LIN {X 0,Y 573.251,Z 441.775,A -85,B 0,C 180,E1 -2241.895,E2 -2241.895} C_VEL
LIN {X 0,Y 573.192,Z 450.436,A -85,B 0,C 180,E1 -2242.603,E2 -2242.603} C_VEL
LIN {X 0,Y 573.159,Z 458.426,A -85,B 0,C 180,E1 -2243.424,E2 -2243.424} C_VEL
LIN {X 0,Y 573.113,Z 464.437,A -85,B 0,C 180,E1 -2244.194,E2 -2244.194} C_VEL
LIN {X 0,Y 572.995,Z 469.99,A -85,B 0,C 180,E1 -2245.075,E2 -2245.075} C_VEL
LIN {X 0,Y 573.036,Z 475.15,A -85,B 0,C 180,E1 -2246.133,E2 -2246.133} C_VEL
LIN {X 0,Y 572.99,Z 477.789,A -85,B 0,C 180,E1 -2246.836,E2 -2246.836} C_VEL
LIN {X 0,Y 572.94,Z 480.683,A -85,B 0,C 180,E1 -2247.891,E2 -2247.891} C_VEL
LIN {X 0,Y 572.944,Z 481.935,A -85,B 0,C 180,E1 -2248.595,E2 -2248.595} C_VEL
LIN {X 0,Y 572.937,Z 482.71,A -85,B 0,C 180,E1 -2249.298,E2 -2249.298} C_VEL
LIN {X 0,Y 572.935,Z 483,A -85,B 0,C 180,E1 -2250,E2 -2250} C_VEL
LIN {X 0,Y 572.937,Z 482.709,A -85,B 0,C 180,E1 -2250.703,E2 -2250.703} C_VEL
LIN {X 0,Y 572.944,Z 481.934,A -85,B 0,C 180,E1 -2251.406,E2 -2251.406} C_VEL
LIN {X 0,Y 572.94,Z 480.68,A -85,B 0,C 180,E1 -2252.109,E2 -2252.109} C_VEL
LIN {X 0,Y 572.99,Z 477.786,A -85,B 0,C 180,E1 -2253.164,E2 -2253.164} C_VEL
LIN {X 0,Y 573.036,Z 475.147,A -85,B 0,C 180,E1 -2253.868,E2 -2253.868} C_VEL
LIN {X 0,Y 572.995,Z 469.984,A -85,B 0,C 180,E1 -2254.926,E2 -2254.926} C_VEL
LIN {X 0,Y 573.138,Z 463.183,A -85,B 0,C 180,E1 -2255.983,E2 -2255.983} C_VEL
LIN {X 0,Y 573.164,Z 455.8,A -85,B 0,C 180,E1 -2256.86,E2 -2256.86} C_VEL
LIN {X 0,Y 573.215,Z 448.402,A -85,B 0,C 180,E1 -2257.574,E2 -2257.574} C_VEL
LIN {X 0,Y 573.278,Z 440.539,A -85,B 0,C 180,E1 -2258.194,E2 -2258.194} C_VEL
LIN {X 0,Y 573.323,Z 430.724,A -85,B 0,C 180,E1 -2258.814,E2 -2258.814} C_VEL
LIN {X 0,Y 573.387,Z 419.295,A -85,B 0,C 180,E1 -2259.347,E2 -2259.347} C_VEL
LIN {X 0,Y 573.48,Z 409.234,A -85,B 0,C 180,E1 -2259.679,E2 -2259.679} C_VEL
LIN {X 0,Y 573.512,Z 400.423,A -85,B 0,C 180,E1 -2259.879,E2 -2259.879} C_VEL
LIN {X 0,Y 573.604,Z 327.515,A -85,B 0,C 180,E1 -2260.808,E2 -2260.808} C_VEL
LIN {X 0,Y 573.152,Z 322.288,A -85,B 0,C 180,E1 -2260.89,E2 -2260.89} C_VEL
LIN {X 0,Y 573.327,Z 305.23,A -85,B 0,C 180,E1 -2263.469,E2 -2263.469} C_VEL
LIN {X 0,Y 573.462,Z 287.427,A -85,B 0,C 180,E1 -2266.189,E2 -2266.189} C_VEL
LIN {X 0,Y 573.63,Z 269.625,A -85,B 0,C 180,E1 -2268.946,E2 -2268.946} C_VEL
LIN {X 0,Y 573.779,Z 252.639,A -85,B 0,C 180,E1 -2271.559,E2 -2271.559} C_VEL
LIN {X 0,Y 573.655,Z 246.517,A -85,B 0,C 180,E1 -2272.511,E2 -2272.511} C_VEL
LIN {X 0,Y 573.209,Z 243.899,A -85,B 0,C 180,E1 -2272.946,E2 -2272.946} C_VEL
LIN {X 0,Y 573.2,Z 243.901,A -85,B 0,C 180,E1 -2275.413,E2 -2275.413} C_VEL
LIN {X 0,Y 573.191,Z 243.894,A -85,B 0,C 180,E1 -2278.018,E2 -2278.018} C_VEL
LIN {X 0,Y 573.2,Z 243.895,A -85,B 0,C 180,E1 -2280.877,E2 -2280.877} C_VEL
LIN {X 0,Y 573.215,Z 243.896,A -85,B 0,C 180,E1 -2283.517,E2 -2283.517} C_VEL
LIN {X 0,Y 573.176,Z 243.895,A -85,B 0,C 180,E1 -2286.055,E2 -2286.055} C_VEL
LIN {X 0,Y 573.175,Z 243.898,A -85,B 0,C 180,E1 -2288.707,E2 -2288.707} C_VEL
LIN {X 0,Y 573.19,Z 243.896,A -85,B 0,C 180,E1 -2291.588,E2 -2291.588} C_VEL
LIN {X 0,Y 573.204,Z 243.896,A -85,B 0,C 180,E1 -2294.673,E2 -2294.673} C_VEL
LIN {X 0,Y 573.2,Z 243.893,A -85,B 0,C 180,E1 -2297.596,E2 -2297.596} C_VEL
LIN {X 0,Y 573.229,Z 243.893,A -85,B 0,C 180,E1 -2300.57,E2 -2300.57} C_VEL
LIN {X 0,Y 573.219,Z 243.896,A -85,B 0,C 180,E1 -2303.075,E2 -2303.075} C_VEL
LIN {X 0,Y 573.232,Z 243.888,A -85,B 0,C 180,E1 -2305.669,E2 -2305.669} C_VEL
LIN {X 0,Y 573.205,Z 243.893,A -85,B 0,C 180,E1 -2308.182,E2 -2308.182} C_VEL
LIN {X 0,Y 573.212,Z 243.899,A -85,B 0,C 180,E1 -2310.631,E2 -2310.631} C_VEL
LIN {X 0,Y 573.194,Z 243.893,A -85,B 0,C 180,E1 -2313.517,E2 -2313.517} C_VEL
LIN {X 0,Y 573.188,Z 243.897,A -85,B 0,C 180,E1 -2316.133,E2 -2316.133} C_VEL
LIN {X 0,Y 573.216,Z 243.892,A -85,B 0,C 180,E1 -2319.172,E2 -2319.172} C_VEL
LIN {X 0,Y 573.195,Z 243.898,A -85,B 0,C 180,E1 -2322.15,E2 -2322.15} C_VEL
LIN {X 0,Y 573.209,Z 243.892,A -85,B 0,C 180,E1 -2325.08,E2 -2325.08} C_VEL
LIN {X 0,Y 573.223,Z 243.893,A -85,B 0,C 180,E1 -2327.97,E2 -2327.97} C_VEL
LIN {X 0,Y 573.2,Z 243.899,A -85,B 0,C 180,E1 -2330.116,E2 -2330.116} C_VEL
LIN {X 0,Y 573.221,Z 243.891,A -85,B 0,C 180,E1 -2332.958,E2 -2332.958} C_VEL
LIN {X 0,Y 573.271,Z 243.884,A -85,B 0,C 180,E1 -2335.077,E2 -2335.077} C_VEL
LIN {X 0,Y 573.307,Z 243.885,A -85,B 0,C 180,E1 -2337.892,E2 -2337.892} C_VEL
LIN {X 0,Y 573.316,Z 243.886,A -85,B 0,C 180,E1 -2340,E2 -2340} C_VEL
LIN {X 0,Y 573.27,Z 243.884,A -85,B 0,C 180,E1 -2342.811,E2 -2342.811} C_VEL
LIN {X 0,Y 573.265,Z 243.888,A -85,B 0,C 180,E1 -2345.629,E2 -2345.629} C_VEL
LIN {X 0,Y 573.234,Z 243.891,A -85,B 0,C 180,E1 -2348.46,E2 -2348.46} C_VEL
LIN {X 0,Y 573.236,Z 243.89,A -85,B 0,C 180,E1 -2351.313,E2 -2351.313} C_VEL
LIN {X 0,Y 573.238,Z 243.89,A -85,B 0,C 180,E1 -2354.406,E2 -2354.406} C_VEL
LIN {X 0,Y 573.193,Z 243.895,A -85,B 0,C 180,E1 -2357.114,E2 -2357.114} C_VEL
LIN {X 0,Y 573.204,Z 243.896,A -85,B 0,C 180,E1 -2360.078,E2 -2360.078} C_VEL
LIN {X 0,Y 573.195,Z 243.894,A -85,B 0,C 180,E1 -2362.34,E2 -2362.34} C_VEL
LIN {X 0,Y 573.194,Z 243.894,A -85,B 0,C 180,E1 -2364.344,E2 -2364.344} C_VEL
LIN {X 0,Y 572.557,Z 243.974,A -85,B 0,C 180,E1 -2364.93,E2 -2364.93} C_VEL
LIN {X 0,Y 569.725,Z 244.332,A -85,B 0,C 180,E1 -2365.882,E2 -2365.882} C_VEL
LIN {X 0,Y 567.305,Z 244.636,A -85,B 0,C 180,E1 -2366.647,E2 -2366.647} C_VEL
LIN {X 0,Y 566.246,Z 244.766,A -85,B 0,C 180,E1 -2367.238,E2 -2367.238} C_VEL
LIN {X 0,Y 566.151,Z 244.776,A -85,B 0,C 180,E1 -2367.439,E2 -2367.439} C_VEL
LIN {X 0,Y 566.149,Z 244.777,A -85,B 0,C 180,E1 -2369.772,E2 -2369.772} C_VEL
LIN {X 0,Y 566.192,Z 244.766,A -85,B 0,C 180,E1 -2372.428,E2 -2372.428} C_VEL
LIN {X 0,Y 566.164,Z 244.773,A -85,B 0,C 180,E1 -2374.987,E2 -2374.987} C_VEL
LIN {X 0,Y 566.189,Z 244.774,A -85,B 0,C 180,E1 -2377.462,E2 -2377.462} C_VEL
LIN {X 0,Y 566.195,Z 244.765,A -85,B 0,C 180,E1 -2380.2,E2 -2380.2} C_VEL
LIN {X 0,Y 566.179,Z 244.774,A -85,B 0,C 180,E1 -2383.056,E2 -2383.056} C_VEL
LIN {X 0,Y 566.156,Z 244.77,A -85,B 0,C 180,E1 -2386.053,E2 -2386.053} C_VEL
LIN {X 0,Y 566.155,Z 244.776,A -85,B 0,C 180,E1 -2388.858,E2 -2388.858} C_VEL
LIN {X 0,Y 566.203,Z 244.768,A -85,B 0,C 180,E1 -2391.443,E2 -2391.443} C_VEL
LIN {X 0,Y 566.141,Z 244.773,A -85,B 0,C 180,E1 -2394.306,E2 -2394.306} C_VEL
LIN {X 0,Y 566.194,Z 244.773,A -85,B 0,C 180,E1 -2396.896,E2 -2396.896} C_VEL
LIN {X 0,Y 566.16,Z 244.772,A -85,B 0,C 180,E1 -2399.406,E2 -2399.406} C_VEL
LIN {X 0,Y 566.149,Z 244.771,A -85,B 0,C 180,E1 -2401.854,E2 -2401.854} C_VEL
LIN {X 0,Y 566.187,Z 244.768,A -85,B 0,C 180,E1 -2404.249,E2 -2404.249} C_VEL
LIN {X 0,Y 566.147,Z 244.773,A -85,B 0,C 180,E1 -2407.367,E2 -2407.367} C_VEL
LIN {X 0,Y 566.171,Z 244.768,A -85,B 0,C 180,E1 -2409.661,E2 -2409.661} C_VEL
LIN {X 0,Y 566.166,Z 244.769,A -85,B 0,C 180,E1 -2411.92,E2 -2411.92} C_VEL
LIN {X 0,Y 566.172,Z 244.839,A -85,B 0,C 180,E1 -2414.198,E2 -2414.198} C_VEL
LIN {X 0,Y 566.045,Z 256.904,A -85,B 0,C 180,E1 -2417.086,E2 -2417.086} C_VEL
LIN {X 0,Y 565.985,Z 265.442,A -85,B 0,C 180,E1 -2419.063,E2 -2419.063} C_VEL
LIN {X 0,Y 566.666,Z 271.419,A -85,B 0,C 180,E1 -2419.152,E2 -2419.152} C_VEL
LIN {X 0,Y 566.539,Z 340.424,A -85,B 0,C 180,E1 -2420.043,E2 -2420.043} C_VEL
LIN {X 0,Y 566.455,Z 350.067,A -85,B 0,C 180,E1 -2420.267,E2 -2420.267} C_VEL
LIN {X 0,Y 566.371,Z 361.605,A -85,B 0,C 180,E1 -2420.671,E2 -2420.671} C_VEL
LIN {X 0,Y 566.299,Z 371.47,A -85,B 0,C 180,E1 -2421.165,E2 -2421.165} C_VEL
LIN {X 0,Y 566.252,Z 379.918,A -85,B 0,C 180,E1 -2421.704,E2 -2421.704} C_VEL
LIN {X 0,Y 566.169,Z 387.886,A -85,B 0,C 180,E1 -2422.331,E2 -2422.331} C_VEL
LIN {X 0,Y 566.099,Z 394.656,A -85,B 0,C 180,E1 -2422.978,E2 -2422.978} C_VEL
LIN {X 0,Y 566.071,Z 399.998,A -85,B 0,C 180,E1 -2423.584,E2 -2423.584} C_VEL
LIN {X 0,Y 566.025,Z 405.309,A -85,B 0,C 180,E1 -2424.299,E2 -2424.299} C_VEL
LIN {X 0,Y 565.917,Z 409.743,A -85,B 0,C 180,E1 -2425.013,E2 -2425.013} C_VEL
LIN {X 0,Y 565.961,Z 413.439,A -85,B 0,C 180,E1 -2425.727,E2 -2425.727} C_VEL
LIN {X 0,Y 565.914,Z 417.641,A -85,B 0,C 180,E1 -2426.796,E2 -2426.796} C_VEL
LIN {X 0,Y 565.842,Z 420.579,A -85,B 0,C 180,E1 -2427.864,E2 -2427.864} C_VEL
LIN {X 0,Y 565.844,Z 421.871,A -85,B 0,C 180,E1 -2428.576,E2 -2428.576} C_VEL
LIN {X 0,Y 565.837,Z 422.688,A -85,B 0,C 180,E1 -2429.288,E2 -2429.288} C_VEL
LIN {X 0,Y 565.837,Z 422.996,A -85,B 0,C 180,E1 -2430,E2 -2430} C_VEL
LIN {X 0,Y 565.838,Z 422.729,A -85,B 0,C 180,E1 -2430.711,E2 -2430.711} C_VEL
LIN {X 0,Y 565.845,Z 421.994,A -85,B 0,C 180,E1 -2431.423,E2 -2431.423} C_VEL
LIN {X 0,Y 565.842,Z 420.785,A -85,B 0,C 180,E1 -2432.135,E2 -2432.135} C_VEL
LIN {X 0,Y 565.913,Z 417.934,A -85,B 0,C 180,E1 -2433.203,E2 -2433.203} C_VEL
LIN {X 0,Y 565.935,Z 415.342,A -85,B 0,C 180,E1 -2433.916,E2 -2433.916} C_VEL
LIN {X 0,Y 565.895,Z 410.232,A -85,B 0,C 180,E1 -2434.987,E2 -2434.987} C_VEL
LIN {X 0,Y 566.057,Z 404.734,A -85,B 0,C 180,E1 -2435.879,E2 -2435.879} C_VEL
LIN {X 0,Y 566.077,Z 397.824,A -85,B 0,C 180,E1 -2436.775,E2 -2436.775} C_VEL
LIN {X 0,Y 566.149,Z 388.913,A -85,B 0,C 180,E1 -2437.668,E2 -2437.668} C_VEL
LIN {X 0,Y 566.267,Z 381.158,A -85,B 0,C 180,E1 -2438.295,E2 -2438.295} C_VEL
LIN {X 0,Y 566.32,Z 372.983,A -85,B 0,C 180,E1 -2438.834,E2 -2438.834} C_VEL
LIN {X 0,Y 566.342,Z 364.464,A -85,B 0,C 180,E1 -2439.283,E2 -2439.283} C_VEL
LIN {X 0,Y 566.439,Z 353.233,A -85,B 0,C 180,E1 -2439.732,E2 -2439.732} C_VEL
LIN {X 0,Y 566.573,Z 341.753,A -85,B 0,C 180,E1 -2440.023,E2 -2440.023} C_VEL
LIN {X 0,Y 566.601,Z 322.559,A -85,B 0,C 180,E1 -2440.293,E2 -2440.293} C_VEL
LIN {X 0,Y 566.545,Z 269.375,A -85,B 0,C 180,E1 -2440.966,E2 -2440.966} C_VEL
LIN {X 0,Y 565.964,Z 265.144,A -85,B 0,C 180,E1 -2441.048,E2 -2441.048} C_VEL
LIN {X 0,Y 566.063,Z 254.223,A -85,B 0,C 180,E1 -2443.644,E2 -2443.644} C_VEL
LIN {X 0,Y 566.154,Z 244.775,A -85,B 0,C 180,E1 -2445.941,E2 -2445.941} C_VEL
LIN {X 0,Y 566.181,Z 244.768,A -85,B 0,C 180,E1 -2448.828,E2 -2448.828} C_VEL
LIN {X 0,Y 566.193,Z 244.773,A -85,B 0,C 180,E1 -2451.416,E2 -2451.416} C_VEL
LIN {X 0,Y 566.151,Z 244.771,A -85,B 0,C 180,E1 -2454.182,E2 -2454.182} C_VEL
LIN {X 0,Y 566.173,Z 244.77,A -85,B 0,C 180,E1 -2456.652,E2 -2456.652} C_VEL
LIN {X 0,Y 566.147,Z 244.773,A -85,B 0,C 180,E1 -2459.771,E2 -2459.771} C_VEL
LIN {X 0,Y 566.188,Z 244.767,A -85,B 0,C 180,E1 -2462.427,E2 -2462.427} C_VEL
LIN {X 0,Y 566.158,Z 244.778,A -85,B 0,C 180,E1 -2464.986,E2 -2464.986} C_VEL
LIN {X 0,Y 566.187,Z 244.77,A -85,B 0,C 180,E1 -2467.461,E2 -2467.461} C_VEL
LIN {X 0,Y 566.201,Z 244.765,A -85,B 0,C 180,E1 -2470.199,E2 -2470.199} C_VEL
LIN {X 0,Y 566.174,Z 244.776,A -85,B 0,C 180,E1 -2473.056,E2 -2473.056} C_VEL
LIN {X 0,Y 566.151,Z 244.771,A -85,B 0,C 180,E1 -2476.053,E2 -2476.053} C_VEL
LIN {X 0,Y 566.145,Z 244.779,A -85,B 0,C 180,E1 -2478.858,E2 -2478.858} C_VEL
LIN {X 0,Y 566.193,Z 244.766,A -85,B 0,C 180,E1 -2481.443,E2 -2481.443} C_VEL
LIN {X 0,Y 566.134,Z 244.777,A -85,B 0,C 180,E1 -2484.306,E2 -2484.306} C_VEL
LIN {X 0,Y 566.187,Z 244.772,A -85,B 0,C 180,E1 -2486.896,E2 -2486.896} C_VEL
LIN {X 0,Y 566.154,Z 244.771,A -85,B 0,C 180,E1 -2489.406,E2 -2489.406} C_VEL
LIN {X 0,Y 566.136,Z 244.774,A -85,B 0,C 180,E1 -2491.853,E2 -2491.853} C_VEL
LIN {X 0,Y 566.183,Z 244.773,A -85,B 0,C 180,E1 -2494.249,E2 -2494.249} C_VEL
LIN {X 0,Y 566.15,Z 244.776,A -85,B 0,C 180,E1 -2496.722,E2 -2496.722} C_VEL
LIN {X 0,Y 566.184,Z 244.769,A -85,B 0,C 180,E1 -2498.901,E2 -2498.901} C_VEL
LIN {X 0,Y 566.176,Z 244.768,A -85,B 0,C 180,E1 -2501.171,E2 -2501.171} C_VEL
LIN {X 0,Y 566.163,Z 244.777,A -85,B 0,C 180,E1 -2504.151,E2 -2504.151} C_VEL
LIN {X 0,Y 566.156,Z 244.778,A -85,B 0,C 180,E1 -2506.358,E2 -2506.358} C_VEL
LIN {X 0,Y 566.205,Z 244.764,A -85,B 0,C 180,E1 -2509.27,E2 -2509.27} C_VEL
LIN {X 0,Y 566.181,Z 244.775,A -85,B 0,C 180,E1 -2512.152,E2 -2512.152} C_VEL
LIN {X 0,Y 566.244,Z 244.759,A -85,B 0,C 180,E1 -2515.016,E2 -2515.016} C_VEL
LIN {X 0,Y 566.274,Z 244.763,A -85,B 0,C 180,E1 -2517.866,E2 -2517.866} C_VEL
LIN {X 0,Y 566.28,Z 244.763,A -85,B 0,C 180,E1 -2520,E2 -2520} C_VEL
LIN {X 0,Y 566.231,Z 244.761,A -85,B 0,C 180,E1 -2522.846,E2 -2522.846} C_VEL
LIN {X 0,Y 566.232,Z 244.768,A -85,B 0,C 180,E1 -2525.699,E2 -2525.699} C_VEL
LIN {X 0,Y 566.179,Z 244.767,A -85,B 0,C 180,E1 -2528.566,E2 -2528.566} C_VEL
LIN {X 0,Y 566.186,Z 244.772,A -85,B 0,C 180,E1 -2531.455,E2 -2531.455} C_VEL
LIN {X 0,Y 566.196,Z 244.765,A -85,B 0,C 180,E1 -2534.494,E2 -2534.494} C_VEL
LIN {X 0,Y 566.15,Z 244.777,A -85,B 0,C 180,E1 -2537.333,E2 -2537.333} C_VEL
LIN {X 0,Y 566.167,Z 244.777,A -85,B 0,C 180,E1 -2539.582,E2 -2539.582} C_VEL
LIN {X 0,Y 566.14,Z 244.776,A -85,B 0,C 180,E1 -2541.865,E2 -2541.865} C_VEL
LIN {X 0,Y 566.145,Z 244.772,A -85,B 0,C 180,E1 -2544.183,E2 -2544.183} C_VEL
LIN {X 0,Y 566.164,Z 244.77,A -85,B 0,C 180,E1 -2546.652,E2 -2546.652} C_VEL
LIN {X 0,Y 566.14,Z 244.775,A -85,B 0,C 180,E1 -2549.772,E2 -2549.772} C_VEL
LIN {X 0,Y 566.184,Z 244.767,A -85,B 0,C 180,E1 -2552.428,E2 -2552.428} C_VEL
LIN {X 0,Y 566.153,Z 244.777,A -85,B 0,C 180,E1 -2554.986,E2 -2554.986} C_VEL
LIN {X 0,Y 566.182,Z 244.771,A -85,B 0,C 180,E1 -2557.462,E2 -2557.462} C_VEL
LIN {X 0,Y 566.16,Z 244.769,A -85,B 0,C 180,E1 -2560.203,E2 -2560.203} C_VEL
LIN {X 0,Y 566.17,Z 244.777,A -85,B 0,C 180,E1 -2563.057,E2 -2563.057} C_VEL
LIN {X 0,Y 566.149,Z 244.77,A -85,B 0,C 180,E1 -2566.054,E2 -2566.054} C_VEL
LIN {X 0,Y 566.139,Z 244.78,A -85,B 0,C 180,E1 -2568.858,E2 -2568.858} C_VEL
LIN {X 0,Y 566.165,Z 244.769,A -85,B 0,C 180,E1 -2571.636,E2 -2571.636} C_VEL
LIN {X 0,Y 566.125,Z 244.776,A -85,B 0,C 180,E1 -2574.306,E2 -2574.306} C_VEL
LIN {X 0,Y 566.156,Z 244.776,A -85,B 0,C 180,E1 -2576.894,E2 -2576.894} C_VEL
LIN {X 0,Y 566.144,Z 244.771,A -85,B 0,C 180,E1 -2579.406,E2 -2579.406} C_VEL
LIN {X 0,Y 566.135,Z 244.773,A -85,B 0,C 180,E1 -2581.854,E2 -2581.854} C_VEL
LIN {X 0,Y 566.167,Z 244.773,A -85,B 0,C 180,E1 -2584.249,E2 -2584.249} C_VEL
LIN {X 0,Y 566.163,Z 244.885,A -85,B 0,C 180,E1 -2586.982,E2 -2586.982} C_VEL
LIN {X 0,Y 566.811,Z 249.814,A -85,B 0,C 180,E1 -2587.78,E2 -2587.78} C_VEL
LIN {X 0,Y 566.655,Z 267.933,A -85,B 0,C 180,E1 -2590.595,E2 -2590.595} C_VEL
LIN {X 0,Y 566.529,Z 284.237,A -85,B 0,C 180,E1 -2593.108,E2 -2593.108} C_VEL
LIN {X 0,Y 566.343,Z 304.048,A -85,B 0,C 180,E1 -2596.18,E2 -2596.18} C_VEL
LIN {X 0,Y 566.126,Z 322.264,A -85,B 0,C 180,E1 -2598.97,E2 -2598.97} C_VEL
LIN {X 0,Y 566.684,Z 329.654,A -85,B 0,C 180,E1 -2599.085,E2 -2599.085} C_VEL
LIN {X 0,Y 566.566,Z 399.163,A -85,B 0,C 180,E1 -2599.977,E2 -2599.977} C_VEL
LIN {X 0,Y 566.464,Z 408.427,A -85,B 0,C 180,E1 -2600.178,E2 -2600.178} C_VEL
LIN {X 0,Y 566.416,Z 416.898,A -85,B 0,C 180,E1 -2600.448,E2 -2600.448} C_VEL
LIN {X 0,Y 566.336,Z 425.403,A -85,B 0,C 180,E1 -2600.807,E2 -2600.807} C_VEL
LIN {X 0,Y 566.317,Z 433.734,A -85,B 0,C 180,E1 -2601.256,E2 -2601.256} C_VEL
LIN {X 0,Y 566.211,Z 441.772,A -85,B 0,C 180,E1 -2601.794,E2 -2601.794} C_VEL
LIN {X 0,Y 566.126,Z 450.436,A -85,B 0,C 180,E1 -2602.511,E2 -2602.511} C_VEL
LIN {X 0,Y 566.087,Z 458.905,A -85,B 0,C 180,E1 -2603.402,E2 -2603.402} C_VEL
LIN {X 0,Y 566.057,Z 464.438,A -85,B 0,C 180,E1 -2604.121,E2 -2604.121} C_VEL
LIN {X 0,Y 565.906,Z 469.991,A -85,B 0,C 180,E1 -2605.013,E2 -2605.013} C_VEL
LIN {X 0,Y 565.943,Z 475.15,A -85,B 0,C 180,E1 -2606.084,E2 -2606.084} C_VEL
LIN {X 0,Y 565.88,Z 478.937,A -85,B 0,C 180,E1 -2607.153,E2 -2607.153} C_VEL
LIN {X 0,Y 565.841,Z 480.683,A -85,B 0,C 180,E1 -2607.865,E2 -2607.865} C_VEL
LIN {X 0,Y 565.844,Z 481.934,A -85,B 0,C 180,E1 -2608.577,E2 -2608.577} C_VEL
LIN {X 0,Y 565.837,Z 482.709,A -85,B 0,C 180,E1 -2609.289,E2 -2609.289} C_VEL
LIN {X 0,Y 565.836,Z 483,A -85,B 0,C 180,E1 -2610,E2 -2610} C_VEL
LIN {X 0,Y 565.837,Z 482.708,A -85,B 0,C 180,E1 -2610.712,E2 -2610.712} C_VEL
LIN {X 0,Y 565.844,Z 481.932,A -85,B 0,C 180,E1 -2611.424,E2 -2611.424} C_VEL
LIN {X 0,Y 565.841,Z 480.681,A -85,B 0,C 180,E1 -2612.136,E2 -2612.136} C_VEL
LIN {X 0,Y 565.912,Z 477.786,A -85,B 0,C 180,E1 -2613.204,E2 -2613.204} C_VEL
LIN {X 0,Y 565.944,Z 475.147,A -85,B 0,C 180,E1 -2613.917,E2 -2613.917} C_VEL
LIN {X 0,Y 565.906,Z 469.984,A -85,B 0,C 180,E1 -2614.988,E2 -2614.988} C_VEL
LIN {X 0,Y 566.082,Z 463.182,A -85,B 0,C 180,E1 -2616.058,E2 -2616.058} C_VEL
LIN {X 0,Y 566.091,Z 456.175,A -85,B 0,C 180,E1 -2616.907,E2 -2616.907} C_VEL
LIN {X 0,Y 566.148,Z 448.399,A -85,B 0,C 180,E1 -2617.669,E2 -2617.669} C_VEL
LIN {X 0,Y 566.261,Z 440.536,A -85,B 0,C 180,E1 -2618.296,E2 -2618.296} C_VEL
LIN {X 0,Y 566.3,Z 430.721,A -85,B 0,C 180,E1 -2618.925,E2 -2618.925} C_VEL
LIN {X 0,Y 566.392,Z 419.297,A -85,B 0,C 180,E1 -2619.463,E2 -2619.463} C_VEL
LIN {X 0,Y 566.463,Z 409.233,A -85,B 0,C 180,E1 -2619.8,E2 -2619.8} C_VEL
LIN {X 0,Y 566.519,Z 400.421,A -85,B 0,C 180,E1 -2620.002,E2 -2620.002} C_VEL
LIN {X 0,Y 566.553,Z 325.807,A -85,B 0,C 180,E1 -2620.966,E2 -2620.966} C_VEL
LIN {X 0,Y 566.1,Z 322.239,A -85,B 0,C 180,E1 -2621.035,E2 -2621.035} C_VEL
LIN {X 0,Y 566.343,Z 304.043,A -85,B 0,C 180,E1 -2623.821,E2 -2623.821} C_VEL
LIN {X 0,Y 566.529,Z 284.234,A -85,B 0,C 180,E1 -2626.892,E2 -2626.892} C_VEL
LIN {X 0,Y 566.648,Z 266.895,A -85,B 0,C 180,E1 -2629.565,E2 -2629.565} C_VEL
LIN {X 0,Y 566.808,Z 249.807,A -85,B 0,C 180,E1 -2632.221,E2 -2632.221} C_VEL
LIN {X 0,Y 566.15,Z 244.779,A -85,B 0,C 180,E1 -2633.044,E2 -2633.044} C_VEL
LIN {X 0,Y 566.17,Z 244.773,A -85,B 0,C 180,E1 -2635.751,E2 -2635.751} C_VEL
LIN {X 0,Y 566.136,Z 244.772,A -85,B 0,C 180,E1 -2638.189,E2 -2638.189} C_VEL
LIN {X 0,Y 566.168,Z 244.774,A -85,B 0,C 180,E1 -2641.072,E2 -2641.072} C_VEL
LIN {X 0,Y 566.176,Z 244.77,A -85,B 0,C 180,E1 -2643.729,E2 -2643.729} C_VEL
LIN {X 0,Y 566.141,Z 244.773,A -85,B 0,C 180,E1 -2646.575,E2 -2646.575} C_VEL
LIN {X 0,Y 566.179,Z 244.769,A -85,B 0,C 180,E1 -2649.681,E2 -2649.681} C_VEL
LIN {X 0,Y 566.146,Z 244.778,A -85,B 0,C 180,E1 -2652.911,E2 -2652.911} C_VEL
LIN {X 0,Y 566.155,Z 244.77,A -85,B 0,C 180,E1 -2655.96,E2 -2655.96} C_VEL
LIN {X 0,Y 566.14,Z 244.78,A -85,B 0,C 180,E1 -2658.857,E2 -2658.857} C_VEL
LIN {X 0,Y 566.18,Z 244.769,A -85,B 0,C 180,E1 -2661.446,E2 -2661.446} C_VEL
LIN {X 0,Y 566.129,Z 244.775,A -85,B 0,C 180,E1 -2664.306,E2 -2664.306} C_VEL
LIN {X 0,Y 566.16,Z 244.777,A -85,B 0,C 180,E1 -2666.894,E2 -2666.894} C_VEL
LIN {X 0,Y 566.147,Z 244.772,A -85,B 0,C 180,E1 -2669.405,E2 -2669.405} C_VEL
LIN {X 0,Y 566.139,Z 244.772,A -85,B 0,C 180,E1 -2671.854,E2 -2671.854} C_VEL
LIN {X 0,Y 566.17,Z 244.772,A -85,B 0,C 180,E1 -2674.249,E2 -2674.249} C_VEL
LIN {X 0,Y 566.146,Z 244.778,A -85,B 0,C 180,E1 -2676.725,E2 -2676.725} C_VEL
LIN {X 0,Y 566.182,Z 244.771,A -85,B 0,C 180,E1 -2678.901,E2 -2678.901} C_VEL
LIN {X 0,Y 566.15,Z 244.772,A -85,B 0,C 180,E1 -2681.92,E2 -2681.92} C_VEL
LIN {X 0,Y 566.152,Z 244.773,A -85,B 0,C 180,E1 -2684.889,E2 -2684.889} C_VEL
LIN {X 0,Y 566.162,Z 244.771,A -85,B 0,C 180,E1 -2687.817,E2 -2687.817} C_VEL
LIN {X 0,Y 566.155,Z 244.775,A -85,B 0,C 180,E1 -2689.992,E2 -2689.992} C_VEL
LIN {X 0,Y 566.183,Z 244.768,A -85,B 0,C 180,E1 -2692.87,E2 -2692.87} C_VEL
LIN {X 0,Y 566.247,Z 244.759,A -85,B 0,C 180,E1 -2695.016,E2 -2695.016} C_VEL
LIN {X 0,Y 566.277,Z 244.76,A -85,B 0,C 180,E1 -2697.866,E2 -2697.866} C_VEL
LIN {X 0,Y 566.285,Z 244.762,A -85,B 0,C 180,E1 -2700,E2 -2700} C_VEL
LIN {X 0,Y 566.238,Z 244.76,A -85,B 0,C 180,E1 -2702.846,E2 -2702.846} C_VEL
LIN {X 0,Y 566.234,Z 244.765,A -85,B 0,C 180,E1 -2705.699,E2 -2705.699} C_VEL
LIN {X 0,Y 566.186,Z 244.768,A -85,B 0,C 180,E1 -2708.566,E2 -2708.566} C_VEL
LIN {X 0,Y 566.194,Z 244.769,A -85,B 0,C 180,E1 -2711.455,E2 -2711.455} C_VEL
LIN {X 0,Y 566.204,Z 244.765,A -85,B 0,C 180,E1 -2714.494,E2 -2714.494} C_VEL
LIN {X 0,Y 566.158,Z 244.773,A -85,B 0,C 180,E1 -2717.333,E2 -2717.333} C_VEL
LIN {X 0,Y 566.175,Z 244.776,A -85,B 0,C 180,E1 -2719.582,E2 -2719.582} C_VEL
LIN {X 0,Y 566.146,Z 244.778,A -85,B 0,C 180,E1 -2721.865,E2 -2721.865} C_VEL
LIN {X 0,Y 566.18,Z 244.769,A -85,B 0,C 180,E1 -2725.021,E2 -2725.021} C_VEL
LIN {X 0,Y 566.151,Z 244.776,A -85,B 0,C 180,E1 -2727.439,E2 -2727.439} C_VEL
LIN {X 0,Y 565.456,Z 244.86,A -85,B 0,C 180,E1 -2728.032,E2 -2728.032} C_VEL
LIN {X 0,Y 562.582,Z 245.218,A -85,B 0,C 180,E1 -2728.996,E2 -2728.996} C_VEL
LIN {X 0,Y 560.183,Z 245.52,A -85,B 0,C 180,E1 -2729.772,E2 -2729.772} C_VEL
LIN {X 0,Y 559.173,Z 245.641,A -85,B 0,C 180,E1 -2730.371,E2 -2730.371} C_VEL
LIN {X 0,Y 559.102,Z 245.649,A -85,B 0,C 180,E1 -2730.574,E2 -2730.574} C_VEL
LIN {X 0,Y 559.148,Z 245.644,A -85,B 0,C 180,E1 -2732.716,E2 -2732.716} C_VEL
LIN {X 0,Y 559.116,Z 245.655,A -85,B 0,C 180,E1 -2735.325,E2 -2735.325} C_VEL
LIN {X 0,Y 559.123,Z 245.647,A -85,B 0,C 180,E1 -2738.018,E2 -2738.018} C_VEL
LIN {X 0,Y 559.15,Z 245.644,A -85,B 0,C 180,E1 -2739.94,E2 -2739.94} C_VEL
LIN {X 0,Y 559.124,Z 245.654,A -85,B 0,C 180,E1 -2743.194,E2 -2743.194} C_VEL
LIN {X 0,Y 559.124,Z 245.648,A -85,B 0,C 180,E1 -2745.764,E2 -2745.764} C_VEL
LIN {X 0,Y 559.101,Z 245.649,A -85,B 0,C 180,E1 -2748.224,E2 -2748.224} C_VEL
LIN {X 0,Y 559.169,Z 245.648,A -85,B 0,C 180,E1 -2751.065,E2 -2751.065} C_VEL
LIN {X 0,Y 559.118,Z 245.648,A -85,B 0,C 180,E1 -2753.787,E2 -2753.787} C_VEL
LIN {X 0,Y 559.145,Z 245.646,A -85,B 0,C 180,E1 -2756.424,E2 -2756.424} C_VEL
LIN {X 0,Y 559.143,Z 245.652,A -85,B 0,C 180,E1 -2758.98,E2 -2758.98} C_VEL
LIN {X 0,Y 559.111,Z 245.648,A -85,B 0,C 180,E1 -2761.63,E2 -2761.63} C_VEL
LIN {X 0,Y 559.156,Z 245.642,A -85,B 0,C 180,E1 -2763.901,E2 -2763.901} C_VEL
LIN {X 0,Y 559.105,Z 245.653,A -85,B 0,C 180,E1 -2767.066,E2 -2767.066} C_VEL
LIN {X 0,Y 559.15,Z 245.644,A -85,B 0,C 180,E1 -2769.394,E2 -2769.394} C_VEL
LIN {X 0,Y 559.117,Z 245.647,A -85,B 0,C 180,E1 -2771.684,E2 -2771.684} C_VEL
LIN {X 0,Y 559.072,Z 245.8,A -85,B 0,C 180,E1 -2774.319,E2 -2774.319} C_VEL
LIN {X 0,Y 558.981,Z 256.889,A -85,B 0,C 180,E1 -2776.92,E2 -2776.92} C_VEL
LIN {X 0,Y 558.897,Z 265.151,A -85,B 0,C 180,E1 -2778.903,E2 -2778.903} C_VEL
LIN {X 0,Y 559.712,Z 272.106,A -85,B 0,C 180,E1 -2779.024,E2 -2779.024} C_VEL
LIN {X 0,Y 559.533,Z 339.16,A -85,B 0,C 180,E1 -2779.895,E2 -2779.895} C_VEL
LIN {X 0,Y 559.478,Z 348.425,A -85,B 0,C 180,E1 -2780.099,E2 -2780.099} C_VEL
LIN {X 0,Y 559.407,Z 356.895,A -85,B 0,C 180,E1 -2780.372,E2 -2780.372} C_VEL
LIN {X 0,Y 559.336,Z 364.461,A -85,B 0,C 180,E1 -2780.69,E2 -2780.69} C_VEL
LIN {X 0,Y 559.296,Z 372.977,A -85,B 0,C 180,E1 -2781.145,E2 -2781.145} C_VEL
LIN {X 0,Y 559.193,Z 381.153,A -85,B 0,C 180,E1 -2781.689,E2 -2781.689} C_VEL
LIN {X 0,Y 559.1,Z 388.911,A -85,B 0,C 180,E1 -2782.324,E2 -2782.324} C_VEL
LIN {X 0,Y 559.017,Z 397.019,A -85,B 0,C 180,E1 -2783.141,E2 -2783.141} C_VEL
LIN {X 0,Y 559.005,Z 404.136,A -85,B 0,C 180,E1 -2784.046,E2 -2784.046} C_VEL
LIN {X 0,Y 558.832,Z 409.746,A -85,B 0,C 180,E1 -2784.949,E2 -2784.949} C_VEL
LIN {X 0,Y 558.893,Z 413.441,A -85,B 0,C 180,E1 -2785.673,E2 -2785.673} C_VEL
LIN {X 0,Y 558.837,Z 417.642,A -85,B 0,C 180,E1 -2786.755,E2 -2786.755} C_VEL
LIN {X 0,Y 558.747,Z 420.579,A -85,B 0,C 180,E1 -2787.837,E2 -2787.837} C_VEL
LIN {X 0,Y 558.743,Z 421.87,A -85,B 0,C 180,E1 -2788.558,E2 -2788.558} C_VEL
LIN {X 0,Y 558.737,Z 422.687,A -85,B 0,C 180,E1 -2789.279,E2 -2789.279} C_VEL
LIN {X 0,Y 558.738,Z 422.996,A -85,B 0,C 180,E1 -2790,E2 -2790} C_VEL
LIN {X 0,Y 558.738,Z 422.728,A -85,B 0,C 180,E1 -2790.72,E2 -2790.72} C_VEL
LIN {X 0,Y 558.745,Z 421.991,A -85,B 0,C 180,E1 -2791.441,E2 -2791.441} C_VEL
LIN {X 0,Y 558.748,Z 420.783,A -85,B 0,C 180,E1 -2792.162,E2 -2792.162} C_VEL
LIN {X 0,Y 558.836,Z 417.932,A -85,B 0,C 180,E1 -2793.244,E2 -2793.244} C_VEL
LIN {X 0,Y 558.852,Z 415.34,A -85,B 0,C 180,E1 -2793.966,E2 -2793.966} C_VEL
LIN {X 0,Y 558.814,Z 410.229,A -85,B 0,C 180,E1 -2795.05,E2 -2795.05} C_VEL
LIN {X 0,Y 559.004,Z 404.731,A -85,B 0,C 180,E1 -2795.953,E2 -2795.953} C_VEL
LIN {X 0,Y 559.024,Z 396.336,A -85,B 0,C 180,E1 -2797.022,E2 -2797.022} C_VEL
LIN {X 0,Y 559.12,Z 388.904,A -85,B 0,C 180,E1 -2797.765,E2 -2797.765} C_VEL
LIN {X 0,Y 559.219,Z 381.146,A -85,B 0,C 180,E1 -2798.4,E2 -2798.4} C_VEL
LIN {X 0,Y 559.283,Z 372.971,A -85,B 0,C 180,E1 -2798.946,E2 -2798.946} C_VEL
LIN {X 0,Y 559.344,Z 364.449,A -85,B 0,C 180,E1 -2799.4,E2 -2799.4} C_VEL
LIN {X 0,Y 559.449,Z 353.215,A -85,B 0,C 180,E1 -2799.855,E2 -2799.855} C_VEL
LIN {X 0,Y 559.592,Z 341.719,A -85,B 0,C 180,E1 -2800.149,E2 -2800.149} C_VEL
LIN {X 0,Y 559.64,Z 322.514,A -85,B 0,C 180,E1 -2800.423,E2 -2800.423} C_VEL
LIN {X 0,Y 559.531,Z 269.605,A -85,B 0,C 180,E1 -2801.102,E2 -2801.102} C_VEL
LIN {X 0,Y 558.905,Z 265.168,A -85,B 0,C 180,E1 -2801.183,E2 -2801.183} C_VEL
LIN {X 0,Y 559.009,Z 252.696,A -85,B 0,C 180,E1 -2804.174,E2 -2804.174} C_VEL
LIN {X 0,Y 559.068,Z 245.66,A -85,B 0,C 180,E1 -2805.82,E2 -2805.82} C_VEL
LIN {X 0,Y 559.112,Z 245.648,A -85,B 0,C 180,E1 -2808.315,E2 -2808.315} C_VEL
LIN {X 0,Y 559.146,Z 245.644,A -85,B 0,C 180,E1 -2810.605,E2 -2810.605} C_VEL
LIN {X 0,Y 559.103,Z 245.653,A -85,B 0,C 180,E1 -2813.718,E2 -2813.718} C_VEL
LIN {X 0,Y 559.151,Z 245.643,A -85,B 0,C 180,E1 -2816.098,E2 -2816.098} C_VEL
LIN {X 0,Y 559.097,Z 245.651,A -85,B 0,C 180,E1 -2818.533,E2 -2818.533} C_VEL
LIN {X 0,Y 559.122,Z 245.654,A -85,B 0,C 180,E1 -2821.269,E2 -2821.269} C_VEL
LIN {X 0,Y 559.148,Z 245.644,A -85,B 0,C 180,E1 -2823.946,E2 -2823.946} C_VEL
LIN {X 0,Y 559.126,Z 245.653,A -85,B 0,C 180,E1 -2827.109,E2 -2827.109} C_VEL
LIN {X 0,Y 559.151,Z 245.643,A -85,B 0,C 180,E1 -2829.94,E2 -2829.94} C_VEL
LIN {X 0,Y 559.119,Z 245.652,A -85,B 0,C 180,E1 -2833.193,E2 -2833.193} C_VEL
LIN {X 0,Y 559.119,Z 245.647,A -85,B 0,C 180,E1 -2835.764,E2 -2835.764} C_VEL
LIN {X 0,Y 559.096,Z 245.652,A -85,B 0,C 180,E1 -2838.223,E2 -2838.223} C_VEL
LIN {X 0,Y 559.162,Z 245.645,A -85,B 0,C 180,E1 -2841.192,E2 -2841.192} C_VEL
LIN {X 0,Y 559.111,Z 245.648,A -85,B 0,C 180,E1 -2843.787,E2 -2843.787} C_VEL
LIN {X 0,Y 559.139,Z 245.651,A -85,B 0,C 180,E1 -2846.423,E2 -2846.423} C_VEL
LIN {X 0,Y 559.139,Z 245.648,A -85,B 0,C 180,E1 -2848.98,E2 -2848.98} C_VEL
LIN {X 0,Y 559.097,Z 245.65,A -85,B 0,C 180,E1 -2851.631,E2 -2851.631} C_VEL
LIN {X 0,Y 559.148,Z 245.645,A -85,B 0,C 180,E1 -2853.901,E2 -2853.901} C_VEL
LIN {X 0,Y 559.099,Z 245.657,A -85,B 0,C 180,E1 -2856.58,E2 -2856.58} C_VEL
LIN {X 0,Y 559.141,Z 245.644,A -85,B 0,C 180,E1 -2859.394,E2 -2859.394} C_VEL
LIN {X 0,Y 559.107,Z 245.65,A -85,B 0,C 180,E1 -2861.684,E2 -2861.684} C_VEL
LIN {X 0,Y 559.121,Z 245.65,A -85,B 0,C 180,E1 -2864.694,E2 -2864.694} C_VEL
LIN {X 0,Y 559.139,Z 245.647,A -85,B 0,C 180,E1 -2867.662,E2 -2867.662} C_VEL
LIN {X 0,Y 559.114,Z 245.653,A -85,B 0,C 180,E1 -2869.864,E2 -2869.864} C_VEL
LIN {X 0,Y 559.142,Z 245.645,A -85,B 0,C 180,E1 -2872.779,E2 -2872.779} C_VEL
LIN {X 0,Y 559.221,Z 245.634,A -85,B 0,C 180,E1 -2874.953,E2 -2874.953} C_VEL
LIN {X 0,Y 559.244,Z 245.638,A -85,B 0,C 180,E1 -2877.839,E2 -2877.839} C_VEL
LIN {X 0,Y 559.248,Z 245.639,A -85,B 0,C 180,E1 -2880,E2 -2880} C_VEL
LIN {X 0,Y 559.2,Z 245.637,A -85,B 0,C 180,E1 -2882.882,E2 -2882.882} C_VEL
LIN {X 0,Y 559.2,Z 245.644,A -85,B 0,C 180,E1 -2885.77,E2 -2885.77} C_VEL
LIN {X 0,Y 559.144,Z 245.644,A -85,B 0,C 180,E1 -2888.675,E2 -2888.675} C_VEL
LIN {X 0,Y 559.148,Z 245.65,A -85,B 0,C 180,E1 -2891.602,E2 -2891.602} C_VEL
LIN {X 0,Y 559.146,Z 245.643,A -85,B 0,C 180,E1 -2894.576,E2 -2894.576} C_VEL
LIN {X 0,Y 559.105,Z 245.657,A -85,B 0,C 180,E1 -2897.559,E2 -2897.559} C_VEL
LIN {X 0,Y 559.13,Z 245.65,A -85,B 0,C 180,E1 -2899.839,E2 -2899.839} C_VEL
LIN {X 0,Y 559.095,Z 245.65,A -85,B 0,C 180,E1 -2902.155,E2 -2902.155} C_VEL
LIN {X 0,Y 559.132,Z 245.651,A -85,B 0,C 180,E1 -2905.178,E2 -2905.178} C_VEL
LIN {X 0,Y 559.094,Z 245.654,A -85,B 0,C 180,E1 -2907.717,E2 -2907.717} C_VEL
LIN {X 0,Y 559.086,Z 245.651,A -85,B 0,C 180,E1 -2910.187,E2 -2910.187} C_VEL
LIN {X 0,Y 559.14,Z 245.646,A -85,B 0,C 180,E1 -2912.716,E2 -2912.716} C_VEL
LIN {X 0,Y 559.106,Z 245.655,A -85,B 0,C 180,E1 -2915.326,E2 -2915.326} C_VEL
LIN {X 0,Y 559.116,Z 245.647,A -85,B 0,C 180,E1 -2918.019,E2 -2918.019} C_VEL
LIN {X 0,Y 559.096,Z 245.655,A -85,B 0,C 180,E1 -2920.818,E2 -2920.818} C_VEL
LIN {X 0,Y 559.1,Z 245.649,A -85,B 0,C 180,E1 -2923.738,E2 -2923.738} C_VEL
LIN {X 0,Y 559.095,Z 245.65,A -85,B 0,C 180,E1 -2926.262,E2 -2926.262} C_VEL
LIN {X 0,Y 559.097,Z 245.654,A -85,B 0,C 180,E1 -2929.183,E2 -2929.183} C_VEL
LIN {X 0,Y 559.117,Z 245.647,A -85,B 0,C 180,E1 -2931.982,E2 -2931.982} C_VEL
LIN {X 0,Y 559.109,Z 245.657,A -85,B 0,C 180,E1 -2934.79,E2 -2934.79} C_VEL
LIN {X 0,Y 559.131,Z 245.646,A -85,B 0,C 180,E1 -2937.368,E2 -2937.368} C_VEL
LIN {X 0,Y 559.091,Z 245.652,A -85,B 0,C 180,E1 -2940.153,E2 -2940.153} C_VEL
LIN {X 0,Y 559.106,Z 245.65,A -85,B 0,C 180,E1 -2943.186,E2 -2943.186} C_VEL
LIN {X 0,Y 559.086,Z 245.652,A -85,B 0,C 180,E1 -2945.492,E2 -2945.492} C_VEL
LIN {X 0,Y 559.144,Z 245.838,A -85,B 0,C 180,E1 -2946.891,E2 -2946.891} C_VEL
LIN {X 0,Y 559.827,Z 250.652,A -85,B 0,C 180,E1 -2947.682,E2 -2947.682} C_VEL
LIN {X 0,Y 559.638,Z 267.695,A -85,B 0,C 180,E1 -2950.366,E2 -2950.366} C_VEL
LIN {X 0,Y 559.502,Z 284.279,A -85,B 0,C 180,E1 -2952.945,E2 -2952.945} C_VEL
LIN {X 0,Y 559.346,Z 304.048,A -85,B 0,C 180,E1 -2956.004,E2 -2956.004} C_VEL
LIN {X 0,Y 559.089,Z 322.259,A -85,B 0,C 180,E1 -2958.828,E2 -2958.828} C_VEL
LIN {X 0,Y 559.719,Z 329.243,A -85,B 0,C 180,E1 -2958.942,E2 -2958.942} C_VEL
LIN {X 0,Y 559.593,Z 399.163,A -85,B 0,C 180,E1 -2959.851,E2 -2959.851} C_VEL
LIN {X 0,Y 559.488,Z 408.426,A -85,B 0,C 180,E1 -2960.054,E2 -2960.054} C_VEL
LIN {X 0,Y 559.424,Z 416.896,A -85,B 0,C 180,E1 -2960.327,E2 -2960.327} C_VEL
LIN {X 0,Y 559.338,Z 425.4,A -85,B 0,C 180,E1 -2960.691,E2 -2960.691} C_VEL
LIN {X 0,Y 559.305,Z 433.731,A -85,B 0,C 180,E1 -2961.146,E2 -2961.146} C_VEL
LIN {X 0,Y 559.199,Z 441.769,A -85,B 0,C 180,E1 -2961.69,E2 -2961.69} C_VEL
LIN {X 0,Y 559.096,Z 450.437,A -85,B 0,C 180,E1 -2962.416,E2 -2962.416} C_VEL
LIN {X 0,Y 559.033,Z 458.735,A -85,B 0,C 180,E1 -2963.296,E2 -2963.296} C_VEL
LIN {X 0,Y 559.004,Z 464.438,A -85,B 0,C 180,E1 -2964.047,E2 -2964.047} C_VEL
LIN {X 0,Y 558.821,Z 469.991,A -85,B 0,C 180,E1 -2964.95,E2 -2964.95} C_VEL
LIN {X 0,Y 558.858,Z 475.151,A -85,B 0,C 180,E1 -2966.034,E2 -2966.034} C_VEL
LIN {X 0,Y 558.803,Z 478.938,A -85,B 0,C 180,E1 -2967.117,E2 -2967.117} C_VEL
LIN {X 0,Y 558.747,Z 480.683,A -85,B 0,C 180,E1 -2967.838,E2 -2967.838} C_VEL
LIN {X 0,Y 558.744,Z 481.932,A -85,B 0,C 180,E1 -2968.559,E2 -2968.559} C_VEL
LIN {X 0,Y 558.737,Z 482.708,A -85,B 0,C 180,E1 -2969.28,E2 -2969.28} C_VEL
LIN {X 0,Y 558.737,Z 483,A -85,B 0,C 180,E1 -2970,E2 -2970} C_VEL
LIN {X 0,Y 558.737,Z 482.707,A -85,B 0,C 180,E1 -2970.721,E2 -2970.721} C_VEL
LIN {X 0,Y 558.744,Z 481.931,A -85,B 0,C 180,E1 -2971.442,E2 -2971.442} C_VEL
LIN {X 0,Y 558.747,Z 480.681,A -85,B 0,C 180,E1 -2972.163,E2 -2972.163} C_VEL
LIN {X 0,Y 558.835,Z 477.786,A -85,B 0,C 180,E1 -2973.245,E2 -2973.245} C_VEL
LIN {X 0,Y 558.858,Z 475.147,A -85,B 0,C 180,E1 -2973.966,E2 -2973.966} C_VEL
LIN {X 0,Y 558.822,Z 469.984,A -85,B 0,C 180,E1 -2975.051,E2 -2975.051} C_VEL
LIN {X 0,Y 559.018,Z 463.181,A -85,B 0,C 180,E1 -2976.135,E2 -2976.135} C_VEL
LIN {X 0,Y 559.036,Z 455.74,A -85,B 0,C 180,E1 -2977.041,E2 -2977.041} C_VEL
LIN {X 0,Y 559.122,Z 448.397,A -85,B 0,C 180,E1 -2977.766,E2 -2977.766} C_VEL
LIN {X 0,Y 559.234,Z 440.533,A -85,B 0,C 180,E1 -2978.401,E2 -2978.401} C_VEL
LIN {X 0,Y 559.289,Z 432.219,A -85,B 0,C 180,E1 -2978.946,E2 -2978.946} C_VEL
LIN {X 0,Y 559.384,Z 421.603,A -85,B 0,C 180,E1 -2979.492,E2 -2979.492} C_VEL
LIN {X 0,Y 559.494,Z 410.064,A -85,B 0,C 180,E1 -2979.901,E2 -2979.901} C_VEL
LIN {X 0,Y 559.529,Z 400.42,A -85,B 0,C 180,E1 -2980.128,E2 -2980.128} C_VEL
LIN {X 0,Y 559.706,Z 330.091,A -85,B 0,C 180,E1 -2981.047,E2 -2981.047} C_VEL
LIN {X 0,Y 559.259,Z 323.907,A -85,B 0,C 180,E1 -2981.135,E2 -2981.135} C_VEL
LIN {X 0,Y 559.06,Z 322.27,A -85,B 0,C 180,E1 -2981.171,E2 -2981.171} C_VEL
LIN {X 0,Y 559.346,Z 304.043,A -85,B 0,C 180,E1 -2983.997,E2 -2983.997} C_VEL
LIN {X 0,Y 559.501,Z 284.275,A -85,B 0,C 180,E1 -2987.055,E2 -2987.055} C_VEL
LIN {X 0,Y 559.647,Z 267.676,A -85,B 0,C 180,E1 -2989.637,E2 -2989.637} C_VEL
LIN {X 0,Y 559.812,Z 250.646,A -85,B 0,C 180,E1 -2992.319,E2 -2992.319} C_VEL
LIN {X 0,Y 559.115,Z 245.655,A -85,B 0,C 180,E1 -2993.146,E2 -2993.146} C_VEL
LIN {X 0,Y 559.139,Z 245.646,A -85,B 0,C 180,E1 -2996.099,E2 -2996.099} C_VEL
LIN {X 0,Y 559.097,Z 245.649,A -85,B 0,C 180,E1 -2998.534,E2 -2998.534} C_VEL
LIN {X 0,Y 559.115,Z 245.656,A -85,B 0,C 180,E1 -3001.268,E2 -3001.268} C_VEL
LIN {X 0,Y 559.136,Z 245.645,A -85,B 0,C 180,E1 -3003.945,E2 -3003.945} C_VEL
LIN {X 0,Y 559.109,Z 245.656,A -85,B 0,C 180,E1 -3007.111,E2 -3007.111} C_VEL
LIN {X 0,Y 559.12,Z 245.646,A -85,B 0,C 180,E1 -3009.937,E2 -3009.937} C_VEL
LIN {X 0,Y 559.109,Z 245.652,A -85,B 0,C 180,E1 -3012.749,E2 -3012.749} C_VEL
LIN {X 0,Y 559.122,Z 245.647,A -85,B 0,C 180,E1 -3015.764,E2 -3015.764} C_VEL
LIN {X 0,Y 559.095,Z 245.65,A -85,B 0,C 180,E1 -3018.224,E2 -3018.224} C_VEL
LIN {X 0,Y 559.134,Z 245.65,A -85,B 0,C 180,E1 -3021.197,E2 -3021.197} C_VEL
LIN {X 0,Y 559.107,Z 245.648,A -85,B 0,C 180,E1 -3023.787,E2 -3023.787} C_VEL
LIN {X 0,Y 559.122,Z 245.65,A -85,B 0,C 180,E1 -3026.422,E2 -3026.422} C_VEL
LIN {X 0,Y 559.133,Z 245.651,A -85,B 0,C 180,E1 -3028.979,E2 -3028.979} C_VEL
LIN {X 0,Y 559.101,Z 245.649,A -85,B 0,C 180,E1 -3031.632,E2 -3031.632} C_VEL
LIN {X 0,Y 559.141,Z 245.644,A -85,B 0,C 180,E1 -3033.901,E2 -3033.901} C_VEL
LIN {X 0,Y 559.09,Z 245.653,A -85,B 0,C 180,E1 -3037.065,E2 -3037.065} C_VEL
LIN {X 0,Y 559.106,Z 245.648,A -85,B 0,C 180,E1 -3039.393,E2 -3039.393} C_VEL
LIN {X 0,Y 559.109,Z 245.656,A -85,B 0,C 180,E1 -3042.442,E2 -3042.442} C_VEL
LIN {X 0,Y 559.152,Z 245.643,A -85,B 0,C 180,E1 -3045.441,E2 -3045.441} C_VEL
LIN {X 0,Y 559.146,Z 245.648,A -85,B 0,C 180,E1 -3048.636,E2 -3048.636} C_VEL
LIN {X 0,Y 559.149,Z 245.643,A -85,B 0,C 180,E1 -3051.325,E2 -3051.325} C_VEL
LIN {X 0,Y 559.204,Z 245.644,A -85,B 0,C 180,E1 -3054.23,E2 -3054.23} C_VEL
LIN {X 0,Y 559.247,Z 245.635,A -85,B 0,C 180,E1 -3057.839,E2 -3057.839} C_VEL
LIN {X 0,Y 559.254,Z 245.638,A -85,B 0,C 180,E1 -3060,E2 -3060} C_VEL
LIN {X 0,Y 559.206,Z 245.636,A -85,B 0,C 180,E1 -3062.882,E2 -3062.882} C_VEL
LIN {X 0,Y 559.204,Z 245.642,A -85,B 0,C 180,E1 -3065.771,E2 -3065.771} C_VEL
LIN {X 0,Y 559.151,Z 245.644,A -85,B 0,C 180,E1 -3068.675,E2 -3068.675} C_VEL
LIN {X 0,Y 559.156,Z 245.648,A -85,B 0,C 180,E1 -3071.602,E2 -3071.602} C_VEL
LIN {X 0,Y 559.154,Z 245.643,A -85,B 0,C 180,E1 -3074.576,E2 -3074.576} C_VEL
LIN {X 0,Y 559.113,Z 245.654,A -85,B 0,C 180,E1 -3077.558,E2 -3077.558} C_VEL
LIN {X 0,Y 559.137,Z 245.652,A -85,B 0,C 180,E1 -3079.839,E2 -3079.839} C_VEL
LIN {X 0,Y 559.102,Z 245.652,A -85,B 0,C 180,E1 -3082.155,E2 -3082.155} C_VEL
LIN {X 0,Y 559.14,Z 245.648,A -85,B 0,C 180,E1 -3085.178,E2 -3085.178} C_VEL
LIN {X 0,Y 559.101,Z 245.656,A -85,B 0,C 180,E1 -3087.717,E2 -3087.717} C_VEL
LIN {X 0,Y 559.102,Z 245.649,A -85,B 0,C 180,E1 -3090.574,E2 -3090.574} C_VEL
LIN {X 0,Y 558.462,Z 245.735,A -85,B 0,C 180,E1 -3091.175,E2 -3091.175} C_VEL
LIN {X 0,Y 555.614,Z 246.087,A -85,B 0,C 180,E1 -3092.152,E2 -3092.152} C_VEL
LIN {X 0,Y 553.196,Z 246.387,A -85,B 0,C 180,E1 -3092.938,E2 -3092.938} C_VEL
LIN {X 0,Y 552.164,Z 246.521,A -85,B 0,C 180,E1 -3093.544,E2 -3093.544} C_VEL
LIN {X 0,Y 552.085,Z 246.524,A -85,B 0,C 180,E1 -3093.75,E2 -3093.75} C_VEL
LIN {X 0,Y 552.098,Z 246.523,A -85,B 0,C 180,E1 -3096.748,E2 -3096.748} C_VEL
LIN {X 0,Y 552.122,Z 246.525,A -85,B 0,C 180,E1 -3099.528,E2 -3099.528} C_VEL
LIN {X 0,Y 552.084,Z 246.524,A -85,B 0,C 180,E1 -3102.43,E2 -3102.43} C_VEL
LIN {X 0,Y 552.075,Z 246.528,A -85,B 0,C 180,E1 -3105.56,E2 -3105.56} C_VEL
LIN {X 0,Y 552.061,Z 246.528,A -85,B 0,C 180,E1 -3108.548,E2 -3108.548} C_VEL
LIN {X 0,Y 552.113,Z 246.524,A -85,B 0,C 180,E1 -3111.41,E2 -3111.41} C_VEL
LIN {X 0,Y 552.071,Z 246.525,A -85,B 0,C 180,E1 -3114.155,E2 -3114.155} C_VEL
LIN {X 0,Y 552.108,Z 246.527,A -85,B 0,C 180,E1 -3117.155,E2 -3117.155} C_VEL
LIN {X 0,Y 552.076,Z 246.526,A -85,B 0,C 180,E1 -3120.233,E2 -3120.233} C_VEL
LIN {X 0,Y 552.093,Z 246.529,A -85,B 0,C 180,E1 -3123.01,E2 -3123.01} C_VEL
LIN {X 0,Y 552.075,Z 246.525,A -85,B 0,C 180,E1 -3125.96,E2 -3125.96} C_VEL
LIN {X 0,Y 552.098,Z 246.525,A -85,B 0,C 180,E1 -3129.119,E2 -3129.119} C_VEL
LIN {X 0,Y 552.08,Z 246.524,A -85,B 0,C 180,E1 -3131.443,E2 -3131.443} C_VEL
LIN {X 0,Y 552.123,Z 246.522,A -85,B 0,C 180,E1 -3134.117,E2 -3134.117} C_VEL
LIN {X 0,Y 551.987,Z 246.714,A -85,B 0,C 180,E1 -3134.397,E2 -3134.397} C_VEL
LIN {X 0,Y 551.896,Z 258.403,A -85,B 0,C 180,E1 -3137.123,E2 -3137.123} C_VEL
LIN {X 0,Y 551.82,Z 265.342,A -85,B 0,C 180,E1 -3138.773,E2 -3138.773} C_VEL
LIN {X 0,Y 552.776,Z 273.049,A -85,B 0,C 180,E1 -3138.894,E2 -3138.894} C_VEL
LIN {X 0,Y 552.558,Z 339.299,A -85,B 0,C 180,E1 -3139.766,E2 -3139.766} C_VEL
LIN {X 0,Y 552.496,Z 348.538,A -85,B 0,C 180,E1 -3139.973,E2 -3139.973} C_VEL
LIN {X 0,Y 552.424,Z 356.983,A -85,B 0,C 180,E1 -3140.249,E2 -3140.249} C_VEL
LIN {X 0,Y 552.339,Z 364.524,A -85,B 0,C 180,E1 -3140.571,E2 -3140.571} C_VEL
LIN {X 0,Y 552.282,Z 373.005,A -85,B 0,C 180,E1 -3141.031,E2 -3141.031} C_VEL
LIN {X 0,Y 552.183,Z 381.157,A -85,B 0,C 180,E1 -3141.583,E2 -3141.583} C_VEL
LIN {X 0,Y 552.07,Z 388.915,A -85,B 0,C 180,E1 -3142.226,E2 -3142.226} C_VEL
LIN {X 0,Y 551.995,Z 395.321,A -85,B 0,C 180,E1 -3142.869,E2 -3142.869} C_VEL
LIN {X 0,Y 551.933,Z 401.074,A -85,B 0,C 180,E1 -3143.558,E2 -3143.558} C_VEL
LIN {X 0,Y 551.87,Z 406.487,A -85,B 0,C 180,E1 -3144.336,E2 -3144.336} C_VEL
LIN {X 0,Y 551.791,Z 411.661,A -85,B 0,C 180,E1 -3145.251,E2 -3145.251} C_VEL
LIN {X 0,Y 551.758,Z 416.457,A -85,B 0,C 180,E1 -3146.348,E2 -3146.348} C_VEL
LIN {X 0,Y 551.731,Z 418.794,A -85,B 0,C 180,E1 -3147.079,E2 -3147.079} C_VEL
LIN {X 0,Y 551.658,Z 420.579,A -85,B 0,C 180,E1 -3147.809,E2 -3147.809} C_VEL
LIN {X 0,Y 551.643,Z 421.869,A -85,B 0,C 180,E1 -3148.54,E2 -3148.54} C_VEL
LIN {X 0,Y 551.637,Z 422.686,A -85,B 0,C 180,E1 -3149.27,E2 -3149.27} C_VEL
LIN {X 0,Y 551.638,Z 422.996,A -85,B 0,C 180,E1 -3150,E2 -3150} C_VEL
LIN {X 0,Y 551.638,Z 422.726,A -85,B 0,C 180,E1 -3150.73,E2 -3150.73} C_VEL
LIN {X 0,Y 551.644,Z 421.989,A -85,B 0,C 180,E1 -3151.46,E2 -3151.46} C_VEL
LIN {X 0,Y 551.658,Z 420.781,A -85,B 0,C 180,E1 -3152.19,E2 -3152.19} C_VEL
LIN {X 0,Y 551.761,Z 417.93,A -85,B 0,C 180,E1 -3153.285,E2 -3153.285} C_VEL
LIN {X 0,Y 551.773,Z 415.337,A -85,B 0,C 180,E1 -3154.017,E2 -3154.017} C_VEL
LIN {X 0,Y 551.738,Z 410.225,A -85,B 0,C 180,E1 -3155.115,E2 -3155.115} C_VEL
LIN {X 0,Y 551.928,Z 404.842,A -85,B 0,C 180,E1 -3156.012,E2 -3156.012} C_VEL
LIN {X 0,Y 551.942,Z 398.139,A -85,B 0,C 180,E1 -3156.911,E2 -3156.911} C_VEL
LIN {X 0,Y 552.066,Z 389.915,A -85,B 0,C 180,E1 -3157.773,E2 -3157.773} C_VEL
LIN {X 0,Y 552.202,Z 382.364,A -85,B 0,C 180,E1 -3158.416,E2 -3158.416} C_VEL
LIN {X 0,Y 552.282,Z 374.472,A -85,B 0,C 180,E1 -3158.968,E2 -3158.968} C_VEL
LIN {X 0,Y 552.321,Z 366.355,A -85,B 0,C 180,E1 -3159.429,E2 -3159.429} C_VEL
LIN {X 0,Y 552.437,Z 358.141,A -85,B 0,C 180,E1 -3159.796,E2 -3159.796} C_VEL
LIN {X 0,Y 552.476,Z 349.303,A -85,B 0,C 180,E1 -3160.096,E2 -3160.096} C_VEL
LIN {X 0,Y 552.623,Z 340.488,A -85,B 0,C 180,E1 -3160.302,E2 -3160.302} C_VEL
LIN {X 0,Y 552.739,Z 287.553,A -85,B 0,C 180,E1 -3161.009,E2 -3161.009} C_VEL
LIN {X 0,Y 552.617,Z 270.623,A -85,B 0,C 180,E1 -3161.231,E2 -3161.231} C_VEL
LIN {X 0,Y 551.855,Z 265.279,A -85,B 0,C 180,E1 -3161.334,E2 -3161.334} C_VEL
LIN {X 0,Y 551.949,Z 252.735,A -85,B 0,C 180,E1 -3164.299,E2 -3164.299} C_VEL
LIN {X 0,Y 551.973,Z 246.545,A -85,B 0,C 180,E1 -3165.745,E2 -3165.745} C_VEL
LIN {X 0,Y 552.075,Z 246.529,A -85,B 0,C 180,E1 -3167.789,E2 -3167.789} C_VEL
LIN {X 0,Y 552.11,Z 246.521,A -85,B 0,C 180,E1 -3170.101,E2 -3170.101} C_VEL
LIN {X 0,Y 552.041,Z 246.529,A -85,B 0,C 180,E1 -3172.453,E2 -3172.453} C_VEL
LIN {X 0,Y 552.08,Z 246.531,A -85,B 0,C 180,E1 -3175.333,E2 -3175.333} C_VEL
LIN {X 0,Y 552.047,Z 246.528,A -85,B 0,C 180,E1 -3178.101,E2 -3178.101} C_VEL
LIN {X 0,Y 552.07,Z 246.527,A -85,B 0,C 180,E1 -3180.611,E2 -3180.611} C_VEL
LIN {X 0,Y 552.1,Z 246.528,A -85,B 0,C 180,E1 -3183.186,E2 -3183.186} C_VEL
LIN {X 0,Y 552.064,Z 246.526,A -85,B 0,C 180,E1 -3185.845,E2 -3185.845} C_VEL
LIN {X 0,Y 552.108,Z 246.524,A -85,B 0,C 180,E1 -3188.589,E2 -3188.589} C_VEL
LIN {X 0,Y 552.056,Z 246.529,A -85,B 0,C 180,E1 -3191.451,E2 -3191.451} C_VEL
LIN {X 0,Y 552.07,Z 246.529,A -85,B 0,C 180,E1 -3194.529,E2 -3194.529} C_VEL
LIN {X 0,Y 552.078,Z 246.525,A -85,B 0,C 180,E1 -3197.59,E2 -3197.59} C_VEL
LIN {X 0,Y 552.117,Z 246.524,A -85,B 0,C 180,E1 -3200.472,E2 -3200.472} C_VEL
LIN {X 0,Y 552.092,Z 246.524,A -85,B 0,C 180,E1 -3203.318,E2 -3203.318} C_VEL
LIN {X 0,Y 552.09,Z 246.524,A -85,B 0,C 180,E1 -3205.936,E2 -3205.936} C_VEL
LIN {X 0,Y 552.099,Z 246.529,A -85,B 0,C 180,E1 -3208.539,E2 -3208.539} C_VEL
LIN {X 0,Y 552.066,Z 246.526,A -85,B 0,C 180,E1 -3211.448,E2 -3211.448} C_VEL
LIN {X 0,Y 552.076,Z 246.532,A -85,B 0,C 180,E1 -3214.353,E2 -3214.353} C_VEL
LIN {X 0,Y 552.045,Z 246.533,A -85,B 0,C 180,E1 -3216.755,E2 -3216.755} C_VEL
LIN {X 0,Y 552.089,Z 246.523,A -85,B 0,C 180,E1 -3219.118,E2 -3219.118} C_VEL
LIN {X 0,Y 552.07,Z 246.525,A -85,B 0,C 180,E1 -3221.442,E2 -3221.442} C_VEL
LIN {X 0,Y 552.066,Z 246.528,A -85,B 0,C 180,E1 -3223.736,E2 -3223.736} C_VEL
LIN {X 0,Y 552.098,Z 246.528,A -85,B 0,C 180,E1 -3226.003,E2 -3226.003} C_VEL
LIN {X 0,Y 552.12,Z 246.519,A -85,B 0,C 180,E1 -3228.992,E2 -3228.992} C_VEL
LIN {X 0,Y 552.102,Z 246.528,A -85,B 0,C 180,E1 -3231.951,E2 -3231.951} C_VEL
LIN {X 0,Y 552.199,Z 246.509,A -85,B 0,C 180,E1 -3234.889,E2 -3234.889} C_VEL
LIN {X 0,Y 552.215,Z 246.514,A -85,B 0,C 180,E1 -3237.812,E2 -3237.812} C_VEL
LIN {X 0,Y 552.216,Z 246.515,A -85,B 0,C 180,E1 -3240,E2 -3240} C_VEL
LIN {X 0,Y 552.168,Z 246.513,A -85,B 0,C 180,E1 -3242.918,E2 -3242.918} C_VEL
LIN {X 0,Y 552.169,Z 246.52,A -85,B 0,C 180,E1 -3245.844,E2 -3245.844} C_VEL
LIN {X 0,Y 552.117,Z 246.519,A -85,B 0,C 180,E1 -3248.786,E2 -3248.786} C_VEL
LIN {X 0,Y 552.093,Z 246.53,A -85,B 0,C 180,E1 -3251.752,E2 -3251.752} C_VEL
LIN {X 0,Y 552.113,Z 246.52,A -85,B 0,C 180,E1 -3254.749,E2 -3254.749} C_VEL
LIN {X 0,Y 552.067,Z 246.531,A -85,B 0,C 180,E1 -3257.79,E2 -3257.79} C_VEL
LIN {X 0,Y 552.085,Z 246.525,A -85,B 0,C 180,E1 -3260.103,E2 -3260.103} C_VEL
LIN {X 0,Y 552.035,Z 246.529,A -85,B 0,C 180,E1 -3262.453,E2 -3262.453} C_VEL
LIN {X 0,Y 552.074,Z 246.532,A -85,B 0,C 180,E1 -3265.334,E2 -3265.334} C_VEL
LIN {X 0,Y 552.041,Z 246.529,A -85,B 0,C 180,E1 -3268.102,E2 -3268.102} C_VEL
LIN {X 0,Y 552.062,Z 246.527,A -85,B 0,C 180,E1 -3270.612,E2 -3270.612} C_VEL
LIN {X 0,Y 552.096,Z 246.529,A -85,B 0,C 180,E1 -3273.187,E2 -3273.187} C_VEL
LIN {X 0,Y 552.06,Z 246.527,A -85,B 0,C 180,E1 -3275.846,E2 -3275.846} C_VEL
LIN {X 0,Y 552.103,Z 246.523,A -85,B 0,C 180,E1 -3278.59,E2 -3278.59} C_VEL
LIN {X 0,Y 552.056,Z 246.53,A -85,B 0,C 180,E1 -3281.452,E2 -3281.452} C_VEL
LIN {X 0,Y 552.069,Z 246.527,A -85,B 0,C 180,E1 -3284.53,E2 -3284.53} C_VEL
LIN {X 0,Y 552.075,Z 246.525,A -85,B 0,C 180,E1 -3287.591,E2 -3287.591} C_VEL
LIN {X 0,Y 552.087,Z 246.526,A -85,B 0,C 180,E1 -3290.47,E2 -3290.47} C_VEL
LIN {X 0,Y 552.047,Z 246.529,A -85,B 0,C 180,E1 -3293.325,E2 -3293.325} C_VEL
LIN {X 0,Y 552.079,Z 246.523,A -85,B 0,C 180,E1 -3295.936,E2 -3295.936} C_VEL
LIN {X 0,Y 552.076,Z 246.53,A -85,B 0,C 180,E1 -3298.538,E2 -3298.538} C_VEL
LIN {X 0,Y 552.066,Z 246.526,A -85,B 0,C 180,E1 -3301.449,E2 -3301.449} C_VEL
LIN {X 0,Y 552.057,Z 246.533,A -85,B 0,C 180,E1 -3304.353,E2 -3304.353} C_VEL
LIN {X 0,Y 552.074,Z 246.564,A -85,B 0,C 180,E1 -3306.757,E2 -3306.757} C_VEL
LIN {X 0,Y 552.851,Z 252.52,A -85,B 0,C 180,E1 -3307.748,E2 -3307.748} C_VEL
LIN {X 0,Y 552.612,Z 269.568,A -85,B 0,C 180,E1 -3310.465,E2 -3310.465} C_VEL
LIN {X 0,Y 552.466,Z 285.585,A -85,B 0,C 180,E1 -3312.988,E2 -3312.988} C_VEL
LIN {X 0,Y 552.287,Z 304.976,A -85,B 0,C 180,E1 -3316.009,E2 -3316.009} C_VEL
LIN {X 0,Y 552.052,Z 322.292,A -85,B 0,C 180,E1 -3318.689,E2 -3318.689} C_VEL
LIN {X 0,Y 552.76,Z 329.365,A -85,B 0,C 180,E1 -3318.803,E2 -3318.803} C_VEL
LIN {X 0,Y 552.619,Z 399.163,A -85,B 0,C 180,E1 -3319.721,E2 -3319.721} C_VEL
LIN {X 0,Y 552.506,Z 408.425,A -85,B 0,C 180,E1 -3319.927,E2 -3319.927} C_VEL
LIN {X 0,Y 552.442,Z 416.894,A -85,B 0,C 180,E1 -3320.204,E2 -3320.204} C_VEL
LIN {X 0,Y 552.326,Z 425.397,A -85,B 0,C 180,E1 -3320.571,E2 -3320.571} C_VEL
LIN {X 0,Y 552.29,Z 433.729,A -85,B 0,C 180,E1 -3321.032,E2 -3321.032} C_VEL
LIN {X 0,Y 552.184,Z 441.766,A -85,B 0,C 180,E1 -3321.584,E2 -3321.584} C_VEL
LIN {X 0,Y 552.068,Z 449.417,A -85,B 0,C 180,E1 -3322.227,E2 -3322.227} C_VEL
LIN {X 0,Y 551.966,Z 457.442,A -85,B 0,C 180,E1 -3323.053,E2 -3323.053} C_VEL
LIN {X 0,Y 551.948,Z 464.517,A -85,B 0,C 180,E1 -3323.983,E2 -3323.983} C_VEL
LIN {X 0,Y 551.743,Z 469.991,A -85,B 0,C 180,E1 -3324.885,E2 -3324.885} C_VEL
LIN {X 0,Y 551.778,Z 475.151,A -85,B 0,C 180,E1 -3325.983,E2 -3325.983} C_VEL
LIN {X 0,Y 551.729,Z 478.938,A -85,B 0,C 180,E1 -3327.08,E2 -3327.08} C_VEL
LIN {X 0,Y 551.657,Z 480.682,A -85,B 0,C 180,E1 -3327.81,E2 -3327.81} C_VEL
LIN {X 0,Y 551.644,Z 481.931,A -85,B 0,C 180,E1 -3328.54,E2 -3328.54} C_VEL
LIN {X 0,Y 551.638,Z 482.707,A -85,B 0,C 180,E1 -3329.27,E2 -3329.27} C_VEL
LIN {X 0,Y 551.637,Z 483,A -85,B 0,C 180,E1 -3330,E2 -3330} C_VEL
LIN {X 0,Y 551.638,Z 482.706,A -85,B 0,C 180,E1 -3330.73,E2 -3330.73} C_VEL
LIN {X 0,Y 551.644,Z 481.929,A -85,B 0,C 180,E1 -3331.46,E2 -3331.46} C_VEL
LIN {X 0,Y 551.657,Z 480.679,A -85,B 0,C 180,E1 -3332.191,E2 -3332.191} C_VEL
LIN {X 0,Y 551.761,Z 477.785,A -85,B 0,C 180,E1 -3333.286,E2 -3333.286} C_VEL
LIN {X 0,Y 551.778,Z 475.147,A -85,B 0,C 180,E1 -3334.017,E2 -3334.017} C_VEL
LIN {X 0,Y 551.743,Z 469.984,A -85,B 0,C 180,E1 -3335.116,E2 -3335.116} C_VEL
LIN {X 0,Y 551.957,Z 463.397,A -85,B 0,C 180,E1 -3336.184,E2 -3336.184} C_VEL
LIN {X 0,Y 551.994,Z 455.738,A -85,B 0,C 180,E1 -3337.131,E2 -3337.131} C_VEL
LIN {X 0,Y 552.078,Z 448.394,A -85,B 0,C 180,E1 -3337.866,E2 -3337.866} C_VEL
LIN {X 0,Y 552.215,Z 440.53,A -85,B 0,C 180,E1 -3338.509,E2 -3338.509} C_VEL
LIN {X 0,Y 552.257,Z 432.217,A -85,B 0,C 180,E1 -3339.061,E2 -3339.061} C_VEL
LIN {X 0,Y 552.393,Z 421.602,A -85,B 0,C 180,E1 -3339.613,E2 -3339.613} C_VEL
LIN {X 0,Y 552.512,Z 410.063,A -85,B 0,C 180,E1 -3340.027,E2 -3340.027} C_VEL
LIN {X 0,Y 552.542,Z 400.419,A -85,B 0,C 180,E1 -3340.258,E2 -3340.258} C_VEL
LIN {X 0,Y 552.776,Z 337.603,A -85,B 0,C 180,E1 -3341.09,E2 -3341.09} C_VEL
LIN {X 0,Y 552.451,Z 325.746,A -85,B 0,C 180,E1 -3341.25,E2 -3341.25} C_VEL
LIN {X 0,Y 552.031,Z 322.228,A -85,B 0,C 180,E1 -3341.322,E2 -3341.322} C_VEL
LIN {X 0,Y 552.307,Z 302.632,A -85,B 0,C 180,E1 -3344.355,E2 -3344.355} C_VEL
LIN {X 0,Y 552.51,Z 282.171,A -85,B 0,C 180,E1 -3347.547,E2 -3347.547} C_VEL
LIN {X 0,Y 552.72,Z 262.466,A -85,B 0,C 180,E1 -3350.662,E2 -3350.662} C_VEL
LIN {X 0,Y 552.699,Z 250.26,A -85,B 0,C 180,E1 -3352.622,E2 -3352.622} C_VEL
LIN {X 0,Y 552.066,Z 246.533,A -85,B 0,C 180,E1 -3353.274,E2 -3353.274} C_VEL
LIN {X 0,Y 552.068,Z 246.526,A -85,B 0,C 180,E1 -3356.46,E2 -3356.46} C_VEL
LIN {X 0,Y 552.035,Z 246.532,A -85,B 0,C 180,E1 -3358.933,E2 -3358.933} C_VEL
LIN {X 0,Y 552.092,Z 246.528,A -85,B 0,C 180,E1 -3361.472,E2 -3361.472} C_VEL
LIN {X 0,Y 552.081,Z 246.523,A -85,B 0,C 180,E1 -3364.162,E2 -3364.162} C_VEL
LIN {X 0,Y 552.05,Z 246.53,A -85,B 0,C 180,E1 -3366.752,E2 -3366.752} C_VEL
LIN {X 0,Y 552.074,Z 246.528,A -85,B 0,C 180,E1 -3369.532,E2 -3369.532} C_VEL
LIN {X 0,Y 552.079,Z 246.524,A -85,B 0,C 180,E1 -3372.431,E2 -3372.431} C_VEL
LIN {X 0,Y 552.073,Z 246.526,A -85,B 0,C 180,E1 -3375.56,E2 -3375.56} C_VEL
LIN {X 0,Y 552.053,Z 246.53,A -85,B 0,C 180,E1 -3378.548,E2 -3378.548} C_VEL
LIN {X 0,Y 552.084,Z 246.525,A -85,B 0,C 180,E1 -3381.408,E2 -3381.408} C_VEL
LIN {X 0,Y 552.056,Z 246.532,A -85,B 0,C 180,E1 -3384.564,E2 -3384.564} C_VEL
LIN {X 0,Y 552.093,Z 246.526,A -85,B 0,C 180,E1 -3387.157,E2 -3387.157} C_VEL
LIN {X 0,Y 552.066,Z 246.526,A -85,B 0,C 180,E1 -3389.959,E2 -3389.959} C_VEL
LIN {X 0,Y 552.075,Z 246.528,A -85,B 0,C 180,E1 -3393.013,E2 -3393.013} C_VEL
LIN {X 0,Y 552.062,Z 246.527,A -85,B 0,C 180,E1 -3395.96,E2 -3395.96} C_VEL
LIN {X 0,Y 552.066,Z 246.527,A -85,B 0,C 180,E1 -3399.118,E2 -3399.118} C_VEL
LIN {X 0,Y 552.045,Z 246.528,A -85,B 0,C 180,E1 -3401.442,E2 -3401.442} C_VEL
LIN {X 0,Y 552.07,Z 246.526,A -85,B 0,C 180,E1 -3403.736,E2 -3403.736} C_VEL
LIN {X 0,Y 552.084,Z 246.527,A -85,B 0,C 180,E1 -3406.754,E2 -3406.754} C_VEL
LIN {X 0,Y 552.125,Z 246.519,A -85,B 0,C 180,E1 -3408.993,E2 -3408.993} C_VEL
LIN {X 0,Y 552.108,Z 246.525,A -85,B 0,C 180,E1 -3411.951,E2 -3411.951} C_VEL
LIN {X 0,Y 552.201,Z 246.51,A -85,B 0,C 180,E1 -3414.889,E2 -3414.889} C_VEL
LIN {X 0,Y 552.218,Z 246.511,A -85,B 0,C 180,E1 -3417.812,E2 -3417.812} C_VEL
LIN {X 0,Y 552.222,Z 246.514,A -85,B 0,C 180,E1 -3420,E2 -3420} C_VEL
LIN {X 0,Y 552.174,Z 246.512,A -85,B 0,C 180,E1 -3422.918,E2 -3422.918} C_VEL
LIN {X 0,Y 552.173,Z 246.519,A -85,B 0,C 180,E1 -3425.844,E2 -3425.844} C_VEL
LIN {X 0,Y 552.124,Z 246.519,A -85,B 0,C 180,E1 -3428.786,E2 -3428.786} C_VEL
LIN {X 0,Y 552.101,Z 246.529,A -85,B 0,C 180,E1 -3431.752,E2 -3431.752} C_VEL
LIN {X 0,Y 552.12,Z 246.519,A -85,B 0,C 180,E1 -3434.749,E2 -3434.749} C_VEL
LIN {X 0,Y 552.075,Z 246.532,A -85,B 0,C 180,E1 -3437.79,E2 -3437.79} C_VEL
LIN {X 0,Y 552.093,Z 246.526,A -85,B 0,C 180,E1 -3440.103,E2 -3440.103} C_VEL
LIN {X 0,Y 552.042,Z 246.529,A -85,B 0,C 180,E1 -3442.453,E2 -3442.453} C_VEL
LIN {X 0,Y 552.084,Z 246.529,A -85,B 0,C 180,E1 -3445.334,E2 -3445.334} C_VEL
LIN {X 0,Y 552.049,Z 246.53,A -85,B 0,C 180,E1 -3448.102,E2 -3448.102} C_VEL
LIN {X 0,Y 552.072,Z 246.525,A -85,B 0,C 180,E1 -3450.611,E2 -3450.611} C_VEL
LIN {X 0,Y 552.104,Z 246.527,A -85,B 0,C 180,E1 -3453.187,E2 -3453.187} C_VEL
LIN {X 0,Y 552.085,Z 246.524,A -85,B 0,C 180,E1 -3453.75,E2 -3453.75} C_VEL
LIN {X 0,Y 551.442,Z 246.606,A -85,B 0,C 180,E1 -3454.358,E2 -3454.358} C_VEL
LIN {X 0,Y 548.632,Z 246.96,A -85,B 0,C 180,E1 -3455.347,E2 -3455.347} C_VEL
LIN {X 0,Y 546.227,Z 247.257,A -85,B 0,C 180,E1 -3456.142,E2 -3456.142} C_VEL
LIN {X 0,Y 545.162,Z 247.388,A -85,B 0,C 180,E1 -3456.756,E2 -3456.756} C_VEL
LIN {X 0,Y 545.06,Z 247.402,A -85,B 0,C 180,E1 -3456.964,E2 -3456.964} C_VEL
LIN {X 0,Y 545.051,Z 247.4,A -85,B 0,C 180,E1 -3460.144,E2 -3460.144} C_VEL
LIN {X 0,Y 545.018,Z 247.41,A -85,B 0,C 180,E1 -3463.113,E2 -3463.113} C_VEL
LIN {X 0,Y 545.028,Z 247.403,A -85,B 0,C 180,E1 -3466.229,E2 -3466.229} C_VEL
LIN {X 0,Y 545.016,Z 247.41,A -85,B 0,C 180,E1 -3468.879,E2 -3468.879} C_VEL
LIN {X 0,Y 545.047,Z 247.401,A -85,B 0,C 180,E1 -3471.762,E2 -3471.762} C_VEL
LIN {X 0,Y 545.025,Z 247.406,A -85,B 0,C 180,E1 -3474.53,E2 -3474.53} C_VEL
LIN {X 0,Y 545.062,Z 247.404,A -85,B 0,C 180,E1 -3477.211,E2 -3477.211} C_VEL
LIN {X 0,Y 545.028,Z 247.403,A -85,B 0,C 180,E1 -3479.808,E2 -3479.808} C_VEL
LIN {X 0,Y 545.037,Z 247.408,A -85,B 0,C 180,E1 -3482.839,E2 -3482.839} C_VEL
LIN {X 0,Y 545.018,Z 247.404,A -85,B 0,C 180,E1 -3485.629,E2 -3485.629} C_VEL
LIN {X 0,Y 545.065,Z 247.4,A -85,B 0,C 180,E1 -3488.181,E2 -3488.181} C_VEL
LIN {X 0,Y 545.104,Z 247.398,A -85,B 0,C 180,E1 -3490.414,E2 -3490.414} C_VEL
LIN {X 0,Y 545.029,Z 247.403,A -85,B 0,C 180,E1 -3493.52,E2 -3493.52} C_VEL
LIN {X 0,Y 544.925,Z 247.517,A -85,B 0,C 180,E1 -3494.429,E2 -3494.429} C_VEL
LIN {X 0,Y 544.842,Z 259.99,A -85,B 0,C 180,E1 -3497.333,E2 -3497.333} C_VEL
LIN {X 0,Y 544.797,Z 265.435,A -85,B 0,C 180,E1 -3498.609,E2 -3498.609} C_VEL
LIN {X 0,Y 545.82,Z 273.641,A -85,B 0,C 180,E1 -3498.752,E2 -3498.752} C_VEL
LIN {X 0,Y 545.593,Z 339.723,A -85,B 0,C 180,E1 -3499.634,E2 -3499.634} C_VEL
LIN {X 0,Y 545.542,Z 348.12,A -85,B 0,C 180,E1 -3499.82,E2 -3499.82} C_VEL
LIN {X 0,Y 545.448,Z 357.389,A -85,B 0,C 180,E1 -3500.123,E2 -3500.123} C_VEL
LIN {X 0,Y 545.358,Z 364.926,A -85,B 0,C 180,E1 -3500.449,E2 -3500.449} C_VEL
LIN {X 0,Y 545.275,Z 373.406,A -85,B 0,C 180,E1 -3500.915,E2 -3500.915} C_VEL
LIN {X 0,Y 545.182,Z 381.54,A -85,B 0,C 180,E1 -3501.474,E2 -3501.474} C_VEL
LIN {X 0,Y 545.04,Z 389.257,A -85,B 0,C 180,E1 -3502.125,E2 -3502.125} C_VEL
LIN {X 0,Y 544.973,Z 395.624,A -85,B 0,C 180,E1 -3502.777,E2 -3502.777} C_VEL
LIN {X 0,Y 544.89,Z 401.914,A -85,B 0,C 180,E1 -3503.55,E2 -3503.55} C_VEL
LIN {X 0,Y 544.762,Z 407.878,A -85,B 0,C 180,E1 -3504.447,E2 -3504.447} C_VEL
LIN {X 0,Y 544.743,Z 413.615,A -85,B 0,C 180,E1 -3505.56,E2 -3505.56} C_VEL
LIN {X 0,Y 544.69,Z 417.777,A -85,B 0,C 180,E1 -3506.671,E2 -3506.671} C_VEL
LIN {X 0,Y 544.573,Z 420.691,A -85,B 0,C 180,E1 -3507.781,E2 -3507.781} C_VEL
LIN {X 0,Y 544.545,Z 421.969,A -85,B 0,C 180,E1 -3508.521,E2 -3508.521} C_VEL
LIN {X 0,Y 544.539,Z 422.779,A -85,B 0,C 180,E1 -3509.26,E2 -3509.26} C_VEL
LIN {X 0,Y 544.54,Z 423.087,A -85,B 0,C 180,E1 -3510,E2 -3510} C_VEL
LIN {X 0,Y 544.54,Z 422.818,A -85,B 0,C 180,E1 -3510.739,E2 -3510.739} C_VEL
LIN {X 0,Y 544.546,Z 422.086,A -85,B 0,C 180,E1 -3511.479,E2 -3511.479} C_VEL
LIN {X 0,Y 544.573,Z 420.888,A -85,B 0,C 180,E1 -3512.218,E2 -3512.218} C_VEL
LIN {X 0,Y 544.688,Z 418.058,A -85,B 0,C 180,E1 -3513.328,E2 -3513.328} C_VEL
LIN {X 0,Y 544.697,Z 415.488,A -85,B 0,C 180,E1 -3514.069,E2 -3514.069} C_VEL
LIN {X 0,Y 544.667,Z 410.422,A -85,B 0,C 180,E1 -3515.182,E2 -3515.182} C_VEL
LIN {X 0,Y 544.904,Z 404.507,A -85,B 0,C 180,E1 -3516.179,E2 -3516.179} C_VEL
LIN {X 0,Y 544.959,Z 396.614,A -85,B 0,C 180,E1 -3517.204,E2 -3517.204} C_VEL
LIN {X 0,Y 545.054,Z 389.223,A -85,B 0,C 180,E1 -3517.967,E2 -3517.967} C_VEL
LIN {X 0,Y 545.186,Z 381.502,A -85,B 0,C 180,E1 -3518.618,E2 -3518.618} C_VEL
LIN {X 0,Y 545.246,Z 373.363,A -85,B 0,C 180,E1 -3519.178,E2 -3519.178} C_VEL
LIN {X 0,Y 545.358,Z 364.868,A -85,B 0,C 180,E1 -3519.644,E2 -3519.644} C_VEL
LIN {X 0,Y 545.475,Z 354.899,A -85,B 0,C 180,E1 -3520.063,E2 -3520.063} C_VEL
LIN {X 0,Y 545.637,Z 343.436,A -85,B 0,C 180,E1 -3520.388,E2 -3520.388} C_VEL
LIN {X 0,Y 545.708,Z 324.722,A -85,B 0,C 180,E1 -3520.668,E2 -3520.668} C_VEL
LIN {X 0,Y 545.713,Z 271.493,A -85,B 0,C 180,E1 -3521.368,E2 -3521.368} C_VEL
LIN {X 0,Y 544.797,Z 265.5,A -85,B 0,C 180,E1 -3521.469,E2 -3521.469} C_VEL
LIN {X 0,Y 544.887,Z 251.749,A -85,B 0,C 180,E1 -3524.68,E2 -3524.68} C_VEL
LIN {X 0,Y 544.922,Z 247.424,A -85,B 0,C 180,E1 -3525.714,E2 -3525.714} C_VEL
LIN {X 0,Y 545.045,Z 247.402,A -85,B 0,C 180,E1 -3528.026,E2 -3528.026} C_VEL
LIN {X 0,Y 545.047,Z 247.4,A -85,B 0,C 180,E1 -3530.373,E2 -3530.373} C_VEL
LIN {X 0,Y 544.986,Z 247.409,A -85,B 0,C 180,E1 -3532.759,E2 -3532.759} C_VEL
LIN {X 0,Y 545.033,Z 247.408,A -85,B 0,C 180,E1 -3535.495,E2 -3535.495} C_VEL
LIN {X 0,Y 545,Z 247.409,A -85,B 0,C 180,E1 -3537.66,E2 -3537.66} C_VEL
LIN {X 0,Y 545.019,Z 247.404,A -85,B 0,C 180,E1 -3540.235,E2 -3540.235} C_VEL
LIN {X 0,Y 545.067,Z 247.405,A -85,B 0,C 180,E1 -3543.06,E2 -3543.06} C_VEL
LIN {X 0,Y 545.014,Z 247.406,A -85,B 0,C 180,E1 -3545.67,E2 -3545.67} C_VEL
LIN {X 0,Y 545.042,Z 247.401,A -85,B 0,C 180,E1 -3548.237,E2 -3548.237} C_VEL
LIN {X 0,Y 545.012,Z 247.411,A -85,B 0,C 180,E1 -3551.12,E2 -3551.12} C_VEL
LIN {X 0,Y 545.027,Z 247.403,A -85,B 0,C 180,E1 -3554.132,E2 -3554.132} C_VEL
LIN {X 0,Y 545.013,Z 247.411,A -85,B 0,C 180,E1 -3556.887,E2 -3556.887} C_VEL
LIN {X 0,Y 545.046,Z 247.4,A -85,B 0,C 180,E1 -3559.855,E2 -3559.855} C_VEL
LIN {X 0,Y 545.059,Z 247.403,A -85,B 0,C 180,E1 -3563.075,E2 -3563.075} C_VEL
LIN {X 0,Y 545.04,Z 247.406,A -85,B 0,C 180,E1 -3566.326,E2 -3566.326} C_VEL
LIN {X 0,Y 545.042,Z 247.405,A -85,B 0,C 180,E1 -3568.95,E2 -3568.95} C_VEL
LIN {X 0,Y 545.027,Z 247.403,A -85,B 0,C 180,E1 -3571.503,E2 -3571.503} C_VEL
LIN {X 0,Y 545.03,Z 247.409,A -85,B 0,C 180,E1 -3574.504,E2 -3574.504} C_VEL
LIN {X 0,Y 544.985,Z 247.408,A -85,B 0,C 180,E1 -3577.24,E2 -3577.24} C_VEL
LIN {X 0,Y 545.096,Z 247.401,A -85,B 0,C 180,E1 -3580.414,E2 -3580.414} C_VEL
LIN {X 0,Y 545.015,Z 247.405,A -85,B 0,C 180,E1 -3583.519,E2 -3583.519} C_VEL
LIN {X 0,Y 545.057,Z 247.402,A -85,B 0,C 180,E1 -3585.819,E2 -3585.819} C_VEL
LIN {X 0,Y 545.066,Z 247.399,A -85,B 0,C 180,E1 -3588.848,E2 -3588.848} C_VEL
LIN {X 0,Y 545.06,Z 247.404,A -85,B 0,C 180,E1 -3591.846,E2 -3591.846} C_VEL
LIN {X 0,Y 545.157,Z 247.387,A -85,B 0,C 180,E1 -3594.822,E2 -3594.822} C_VEL
LIN {X 0,Y 545.185,Z 247.389,A -85,B 0,C 180,E1 -3597.784,E2 -3597.784} C_VEL
LIN {X 0,Y 545.185,Z 247.39,A -85,B 0,C 180,E1 -3600,E2 -3600} C_VEL
LIN {X 0,Y 545.136,Z 247.389,A -85,B 0,C 180,E1 -3602.956,E2 -3602.956} C_VEL
LIN {X 0,Y 545.119,Z 247.399,A -85,B 0,C 180,E1 -3605.92,E2 -3605.92} C_VEL
LIN {X 0,Y 545.06,Z 247.399,A -85,B 0,C 180,E1 -3608.901,E2 -3608.901} C_VEL
LIN {X 0,Y 545.058,Z 247.404,A -85,B 0,C 180,E1 -3611.906,E2 -3611.906} C_VEL
LIN {X 0,Y 545.069,Z 247.398,A -85,B 0,C 180,E1 -3614.944,E2 -3614.944} C_VEL
LIN {X 0,Y 545.036,Z 247.404,A -85,B 0,C 180,E1 -3618.027,E2 -3618.027} C_VEL
LIN {X 0,Y 545.023,Z 247.403,A -85,B 0,C 180,E1 -3620.375,E2 -3620.375} C_VEL
LIN {X 0,Y 544.981,Z 247.409,A -85,B 0,C 180,E1 -3622.76,E2 -3622.76} C_VEL
LIN {X 0,Y 545.025,Z 247.41,A -85,B 0,C 180,E1 -3625.495,E2 -3625.495} C_VEL
LIN {X 0,Y 545.025,Z 247.403,A -85,B 0,C 180,E1 -3628.497,E2 -3628.497} C_VEL
LIN {X 0,Y 545.038,Z 247.404,A -85,B 0,C 180,E1 -3631.676,E2 -3631.676} C_VEL
LIN {X 0,Y 545.037,Z 247.402,A -85,B 0,C 180,E1 -3634.566,E2 -3634.566} C_VEL
LIN {X 0,Y 545.012,Z 247.411,A -85,B 0,C 180,E1 -3637.306,E2 -3637.306} C_VEL
LIN {X 0,Y 545.027,Z 247.402,A -85,B 0,C 180,E1 -3640.146,E2 -3640.146} C_VEL
LIN {X 0,Y 545.011,Z 247.412,A -85,B 0,C 180,E1 -3643.113,E2 -3643.113} C_VEL
LIN {X 0,Y 545.02,Z 247.403,A -85,B 0,C 180,E1 -3646.229,E2 -3646.229} C_VEL
LIN {X 0,Y 545.009,Z 247.413,A -85,B 0,C 180,E1 -3648.879,E2 -3648.879} C_VEL
LIN {X 0,Y 545.035,Z 247.401,A -85,B 0,C 180,E1 -3651.866,E2 -3651.866} C_VEL
LIN {X 0,Y 545.013,Z 247.409,A -85,B 0,C 180,E1 -3654.53,E2 -3654.53} C_VEL
LIN {X 0,Y 545.045,Z 247.402,A -85,B 0,C 180,E1 -3657.211,E2 -3657.211} C_VEL
LIN {X 0,Y 545.012,Z 247.403,A -85,B 0,C 180,E1 -3659.808,E2 -3659.808} C_VEL
LIN {X 0,Y 544.992,Z 247.412,A -85,B 0,C 180,E1 -3662.339,E2 -3662.339} C_VEL
LIN {X 0,Y 545.018,Z 247.411,A -85,B 0,C 180,E1 -3664.816,E2 -3664.816} C_VEL
LIN {X 0,Y 545.036,Z 247.56,A -85,B 0,C 180,E1 -3666.666,E2 -3666.666} C_VEL
LIN {X 0,Y 545.87,Z 253.805,A -85,B 0,C 180,E1 -3667.719,E2 -3667.719} C_VEL
LIN {X 0,Y 545.6,Z 270.613,A -85,B 0,C 180,E1 -3670.433,E2 -3670.433} C_VEL
LIN {X 0,Y 545.429,Z 286.41,A -85,B 0,C 180,E1 -3672.954,E2 -3672.954} C_VEL
LIN {X 0,Y 545.21,Z 305.792,A -85,B 0,C 180,E1 -3676.014,E2 -3676.014} C_VEL
LIN {X 0,Y 544.974,Z 322.042,A -85,B 0,C 180,E1 -3678.55,E2 -3678.55} C_VEL
LIN {X 0,Y 545.772,Z 330.719,A -85,B 0,C 180,E1 -3678.68,E2 -3678.68} C_VEL
LIN {X 0,Y 545.657,Z 398.918,A -85,B 0,C 180,E1 -3679.589,E2 -3679.589} C_VEL
LIN {X 0,Y 545.527,Z 408.195,A -85,B 0,C 180,E1 -3679.797,E2 -3679.797} C_VEL
LIN {X 0,Y 545.437,Z 416.688,A -85,B 0,C 180,E1 -3680.077,E2 -3680.077} C_VEL
LIN {X 0,Y 545.303,Z 425.219,A -85,B 0,C 180,E1 -3680.449,E2 -3680.449} C_VEL
LIN {X 0,Y 545.247,Z 433.591,A -85,B 0,C 180,E1 -3680.916,E2 -3680.916} C_VEL
LIN {X 0,Y 545.155,Z 441.67,A -85,B 0,C 180,E1 -3681.475,E2 -3681.475} C_VEL
LIN {X 0,Y 545.009,Z 450.392,A -85,B 0,C 180,E1 -3682.219,E2 -3682.219} C_VEL
LIN {X 0,Y 544.902,Z 459.083,A -85,B 0,C 180,E1 -3683.167,E2 -3683.167} C_VEL
LIN {X 0,Y 544.844,Z 465.612,A -85,B 0,C 180,E1 -3684.077,E2 -3684.077} C_VEL
LIN {X 0,Y 544.671,Z 469.991,A -85,B 0,C 180,E1 -3684.818,E2 -3684.818} C_VEL
LIN {X 0,Y 544.701,Z 475.151,A -85,B 0,C 180,E1 -3685.931,E2 -3685.931} C_VEL
LIN {X 0,Y 544.658,Z 478.939,A -85,B 0,C 180,E1 -3687.042,E2 -3687.042} C_VEL
LIN {X 0,Y 544.572,Z 480.681,A -85,B 0,C 180,E1 -3687.782,E2 -3687.782} C_VEL
LIN {X 0,Y 544.545,Z 481.929,A -85,B 0,C 180,E1 -3688.521,E2 -3688.521} C_VEL
LIN {X 0,Y 544.538,Z 482.706,A -85,B 0,C 180,E1 -3689.261,E2 -3689.261} C_VEL
LIN {X 0,Y 544.538,Z 483,A -85,B 0,C 180,E1 -3690,E2 -3690} C_VEL
LIN {X 0,Y 544.538,Z 482.705,A -85,B 0,C 180,E1 -3690.74,E2 -3690.74} C_VEL
LIN {X 0,Y 544.545,Z 481.927,A -85,B 0,C 180,E1 -3691.479,E2 -3691.479} C_VEL
LIN {X 0,Y 544.572,Z 480.678,A -85,B 0,C 180,E1 -3692.219,E2 -3692.219} C_VEL
LIN {X 0,Y 544.688,Z 477.785,A -85,B 0,C 180,E1 -3693.329,E2 -3693.329} C_VEL
LIN {X 0,Y 544.701,Z 475.147,A -85,B 0,C 180,E1 -3694.07,E2 -3694.07} C_VEL
LIN {X 0,Y 544.671,Z 469.984,A -85,B 0,C 180,E1 -3695.183,E2 -3695.183} C_VEL
LIN {X 0,Y 544.88,Z 463.956,A -85,B 0,C 180,E1 -3696.183,E2 -3696.183} C_VEL
LIN {X 0,Y 544.92,Z 457.43,A -85,B 0,C 180,E1 -3697.038,E2 -3697.038} C_VEL
LIN {X 0,Y 545.018,Z 449.364,A -85,B 0,C 180,E1 -3697.875,E2 -3697.875} C_VEL
LIN {X 0,Y 545.155,Z 441.664,A -85,B 0,C 180,E1 -3698.526,E2 -3698.526} C_VEL
LIN {X 0,Y 545.248,Z 433.579,A -85,B 0,C 180,E1 -3699.085,E2 -3699.085} C_VEL
LIN {X 0,Y 545.303,Z 425.205,A -85,B 0,C 180,E1 -3699.552,E2 -3699.552} C_VEL
LIN {X 0,Y 545.438,Z 416.671,A -85,B 0,C 180,E1 -3699.924,E2 -3699.924} C_VEL
LIN {X 0,Y 545.531,Z 406.503,A -85,B 0,C 180,E1 -3700.25,E2 -3700.25} C_VEL
LIN {X 0,Y 545.634,Z 394.777,A -85,B 0,C 180,E1 -3700.483,E2 -3700.483} C_VEL
LIN {X 0,Y 545.692,Z 327.896,A -85,B 0,C 180,E1 -3701.359,E2 -3701.359} C_VEL
LIN {X 0,Y 544.976,Z 321.865,A -85,B 0,C 180,E1 -3701.471,E2 -3701.471} C_VEL
LIN {X 0,Y 545.245,Z 302.523,A -85,B 0,C 180,E1 -3704.5,E2 -3704.5} C_VEL
LIN {X 0,Y 545.494,Z 282.158,A -85,B 0,C 180,E1 -3707.721,E2 -3707.721} C_VEL
LIN {X 0,Y 545.715,Z 263.306,A -85,B 0,C 180,E1 -3710.742,E2 -3710.742} C_VEL
LIN {X 0,Y 545.798,Z 252.333,A -85,B 0,C 180,E1 -3712.525,E2 -3712.525} C_VEL
LIN {X 0,Y 545.036,Z 247.409,A -85,B 0,C 180,E1 -3713.36,E2 -3713.36} C_VEL
LIN {X 0,Y 545.027,Z 247.405,A -85,B 0,C 180,E1 -3716.004,E2 -3716.004} C_VEL
LIN {X 0,Y 545.015,Z 247.404,A -85,B 0,C 180,E1 -3718.734,E2 -3718.734} C_VEL
LIN {X 0,Y 545.042,Z 247.404,A -85,B 0,C 180,E1 -3721.676,E2 -3721.676} C_VEL
LIN {X 0,Y 545.037,Z 247.401,A -85,B 0,C 180,E1 -3724.567,E2 -3724.567} C_VEL
LIN {X 0,Y 545.002,Z 247.412,A -85,B 0,C 180,E1 -3727.307,E2 -3727.307} C_VEL
LIN {X 0,Y 545.027,Z 247.402,A -85,B 0,C 180,E1 -3730.146,E2 -3730.146} C_VEL
LIN {X 0,Y 544.998,Z 247.413,A -85,B 0,C 180,E1 -3733.115,E2 -3733.115} C_VEL
LIN {X 0,Y 545.029,Z 247.402,A -85,B 0,C 180,E1 -3735.868,E2 -3735.868} C_VEL
LIN {X 0,Y 545.003,Z 247.413,A -85,B 0,C 180,E1 -3738.878,E2 -3738.878} C_VEL
LIN {X 0,Y 545.024,Z 247.402,A -85,B 0,C 180,E1 -3741.868,E2 -3741.868} C_VEL
LIN {X 0,Y 545.016,Z 247.408,A -85,B 0,C 180,E1 -3744.53,E2 -3744.53} C_VEL
LIN {X 0,Y 545.049,Z 247.403,A -85,B 0,C 180,E1 -3747.21,E2 -3747.21} C_VEL
LIN {X 0,Y 545.016,Z 247.404,A -85,B 0,C 180,E1 -3749.808,E2 -3749.808} C_VEL
LIN {X 0,Y 544.997,Z 247.41,A -85,B 0,C 180,E1 -3752.339,E2 -3752.339} C_VEL
LIN {X 0,Y 545.021,Z 247.409,A -85,B 0,C 180,E1 -3754.816,E2 -3754.816} C_VEL
LIN {X 0,Y 544.987,Z 247.408,A -85,B 0,C 180,E1 -3757.24,E2 -3757.24} C_VEL
LIN {X 0,Y 545.003,Z 247.405,A -85,B 0,C 180,E1 -3759.624,E2 -3759.624} C_VEL
LIN {X 0,Y 545.03,Z 247.407,A -85,B 0,C 180,E1 -3762.748,E2 -3762.748} C_VEL
LIN {X 0,Y 545.048,Z 247.401,A -85,B 0,C 180,E1 -3765.819,E2 -3765.819} C_VEL
LIN {X 0,Y 545.071,Z 247.399,A -85,B 0,C 180,E1 -3768.848,E2 -3768.848} C_VEL
LIN {X 0,Y 545.065,Z 247.401,A -85,B 0,C 180,E1 -3771.846,E2 -3771.846} C_VEL
LIN {X 0,Y 545.159,Z 247.388,A -85,B 0,C 180,E1 -3774.823,E2 -3774.823} C_VEL
LIN {X 0,Y 545.189,Z 247.386,A -85,B 0,C 180,E1 -3777.784,E2 -3777.784} C_VEL
LIN {X 0,Y 545.191,Z 247.39,A -85,B 0,C 180,E1 -3780,E2 -3780} C_VEL
LIN {X 0,Y 545.142,Z 247.388,A -85,B 0,C 180,E1 -3782.956,E2 -3782.956} C_VEL
LIN {X 0,Y 545.124,Z 247.398,A -85,B 0,C 180,E1 -3785.92,E2 -3785.92} C_VEL
LIN {X 0,Y 545.067,Z 247.398,A -85,B 0,C 180,E1 -3788.901,E2 -3788.901} C_VEL
LIN {X 0,Y 545.065,Z 247.405,A -85,B 0,C 180,E1 -3791.906,E2 -3791.906} C_VEL
LIN {X 0,Y 545.076,Z 247.397,A -85,B 0,C 180,E1 -3794.944,E2 -3794.944} C_VEL
LIN {X 0,Y 545.044,Z 247.406,A -85,B 0,C 180,E1 -3798.027,E2 -3798.027} C_VEL
LIN {X 0,Y 545.03,Z 247.403,A -85,B 0,C 180,E1 -3800.375,E2 -3800.375} C_VEL
LIN {X 0,Y 544.988,Z 247.408,A -85,B 0,C 180,E1 -3802.76,E2 -3802.76} C_VEL
LIN {X 0,Y 545.036,Z 247.409,A -85,B 0,C 180,E1 -3805.495,E2 -3805.495} C_VEL
LIN {X 0,Y 545.033,Z 247.402,A -85,B 0,C 180,E1 -3808.496,E2 -3808.496} C_VEL
LIN {X 0,Y 545.045,Z 247.407,A -85,B 0,C 180,E1 -3811.676,E2 -3811.676} C_VEL
LIN {X 0,Y 545.046,Z 247.401,A -85,B 0,C 180,E1 -3814.566,E2 -3814.566} C_VEL
LIN {X 0,Y 545.06,Z 247.402,A -85,B 0,C 180,E1 -3816.964,E2 -3816.964} C_VEL
LIN {X 0,Y 544.349,Z 247.494,A -85,B 0,C 180,E1 -3817.581,E2 -3817.581} C_VEL
LIN {X 0,Y 541.483,Z 247.85,A -85,B 0,C 180,E1 -3818.582,E2 -3818.582} C_VEL
LIN {X 0,Y 539.088,Z 248.149,A -85,B 0,C 180,E1 -3819.387,E2 -3819.387} C_VEL
LIN {X 0,Y 538.063,Z 248.271,A -85,B 0,C 180,E1 -3820.009,E2 -3820.009} C_VEL
LIN {X 0,Y 537.98,Z 248.281,A -85,B 0,C 180,E1 -3820.22,E2 -3820.22} C_VEL
LIN {X 0,Y 537.971,Z 248.287,A -85,B 0,C 180,E1 -3822.981,E2 -3822.981} C_VEL
LIN {X 0,Y 538.002,Z 248.279,A -85,B 0,C 180,E1 -3825.929,E2 -3825.929} C_VEL
LIN {X 0,Y 538.002,Z 248.285,A -85,B 0,C 180,E1 -3829.259,E2 -3829.259} C_VEL
LIN {X 0,Y 537.987,Z 248.28,A -85,B 0,C 180,E1 -3832.122,E2 -3832.122} C_VEL
LIN {X 0,Y 537.987,Z 248.286,A -85,B 0,C 180,E1 -3834.915,E2 -3834.915} C_VEL
LIN {X 0,Y 538.012,Z 248.278,A -85,B 0,C 180,E1 -3837.617,E2 -3837.617} C_VEL
LIN {X 0,Y 537.981,Z 248.282,A -85,B 0,C 180,E1 -3840.236,E2 -3840.236} C_VEL
LIN {X 0,Y 538.009,Z 248.283,A -85,B 0,C 180,E1 -3842.793,E2 -3842.793} C_VEL
LIN {X 0,Y 537.981,Z 248.283,A -85,B 0,C 180,E1 -3845.289,E2 -3845.289} C_VEL
LIN {X 0,Y 538.012,Z 248.278,A -85,B 0,C 180,E1 -3848.043,E2 -3848.043} C_VEL
LIN {X 0,Y 538.008,Z 248.282,A -85,B 0,C 180,E1 -3850.939,E2 -3850.939} C_VEL
LIN {X 0,Y 537.974,Z 248.283,A -85,B 0,C 180,E1 -3853.297,E2 -3853.297} C_VEL
LIN {X 0,Y 537.89,Z 248.361,A -85,B 0,C 180,E1 -3854.463,E2 -3854.463} C_VEL
LIN {X 0,Y 537.795,Z 261.675,A -85,B 0,C 180,E1 -3857.547,E2 -3857.547} C_VEL
LIN {X 0,Y 537.75,Z 265.656,A -85,B 0,C 180,E1 -3858.467,E2 -3858.467} C_VEL
LIN {X 0,Y 538.853,Z 273.107,A -85,B 0,C 180,E1 -3858.592,E2 -3858.592} C_VEL
LIN {X 0,Y 538.632,Z 340.146,A -85,B 0,C 180,E1 -3859.498,E2 -3859.498} C_VEL
LIN {X 0,Y 538.573,Z 348.532,A -85,B 0,C 180,E1 -3859.687,E2 -3859.687} C_VEL
LIN {X 0,Y 538.474,Z 357.796,A -85,B 0,C 180,E1 -3859.994,E2 -3859.994} C_VEL
LIN {X 0,Y 538.381,Z 365.329,A -85,B 0,C 180,E1 -3860.324,E2 -3860.324} C_VEL
LIN {X 0,Y 538.283,Z 373.806,A -85,B 0,C 180,E1 -3860.796,E2 -3860.796} C_VEL
LIN {X 0,Y 538.175,Z 381.939,A -85,B 0,C 180,E1 -3861.362,E2 -3861.362} C_VEL
LIN {X 0,Y 538.032,Z 389.654,A -85,B 0,C 180,E1 -3862.022,E2 -3862.022} C_VEL
LIN {X 0,Y 537.936,Z 396.019,A -85,B 0,C 180,E1 -3862.681,E2 -3862.681} C_VEL
LIN {X 0,Y 537.846,Z 402.741,A -85,B 0,C 180,E1 -3863.523,E2 -3863.523} C_VEL
LIN {X 0,Y 537.655,Z 409.387,A -85,B 0,C 180,E1 -3864.562,E2 -3864.562} C_VEL
LIN {X 0,Y 537.681,Z 414.008,A -85,B 0,C 180,E1 -3865.502,E2 -3865.502} C_VEL
LIN {X 0,Y 537.6,Z 416.997,A -85,B 0,C 180,E1 -3866.252,E2 -3866.252} C_VEL
LIN {X 0,Y 537.592,Z 419.311,A -85,B 0,C 180,E1 -3867.002,E2 -3867.002} C_VEL
LIN {X 0,Y 537.491,Z 421.083,A -85,B 0,C 180,E1 -3867.752,E2 -3867.752} C_VEL
LIN {X 0,Y 537.457,Z 422.361,A -85,B 0,C 180,E1 -3868.501,E2 -3868.501} C_VEL
LIN {X 0,Y 537.45,Z 423.171,A -85,B 0,C 180,E1 -3869.25,E2 -3869.25} C_VEL
LIN {X 0,Y 537.451,Z 423.478,A -85,B 0,C 180,E1 -3870,E2 -3870} C_VEL
LIN {X 0,Y 537.451,Z 423.209,A -85,B 0,C 180,E1 -3870.749,E2 -3870.749} C_VEL
LIN {X 0,Y 537.458,Z 422.477,A -85,B 0,C 180,E1 -3871.498,E2 -3871.498} C_VEL
LIN {X 0,Y 537.491,Z 421.278,A -85,B 0,C 180,E1 -3872.248,E2 -3872.248} C_VEL
LIN {X 0,Y 537.617,Z 418.447,A -85,B 0,C 180,E1 -3873.372,E2 -3873.372} C_VEL
LIN {X 0,Y 537.626,Z 415.877,A -85,B 0,C 180,E1 -3874.123,E2 -3874.123} C_VEL
LIN {X 0,Y 537.605,Z 410.81,A -85,B 0,C 180,E1 -3875.25,E2 -3875.25} C_VEL
LIN {X 0,Y 537.844,Z 405.077,A -85,B 0,C 180,E1 -3876.232,E2 -3876.232} C_VEL
LIN {X 0,Y 537.883,Z 398.496,A -85,B 0,C 180,E1 -3877.13,E2 -3877.13} C_VEL
LIN {X 0,Y 538.024,Z 390.622,A -85,B 0,C 180,E1 -3877.977,E2 -3877.977} C_VEL
LIN {X 0,Y 538.185,Z 383.107,A -85,B 0,C 180,E1 -3878.637,E2 -3878.637} C_VEL
LIN {X 0,Y 538.288,Z 375.236,A -85,B 0,C 180,E1 -3879.203,E2 -3879.203} C_VEL
LIN {X 0,Y 538.375,Z 367.112,A -85,B 0,C 180,E1 -3879.675,E2 -3879.675} C_VEL
LIN {X 0,Y 538.491,Z 358.892,A -85,B 0,C 180,E1 -3880.053,E2 -3880.053} C_VEL
LIN {X 0,Y 538.533,Z 350.043,A -85,B 0,C 180,E1 -3880.361,E2 -3880.361} C_VEL
LIN {X 0,Y 538.708,Z 341.204,A -85,B 0,C 180,E1 -3880.571,E2 -3880.571} C_VEL
LIN {X 0,Y 538.795,Z 289.333,A -85,B 0,C 180,E1 -3881.283,E2 -3881.283} C_VEL
LIN {X 0,Y 538.734,Z 271.84,A -85,B 0,C 180,E1 -3881.517,E2 -3881.517} C_VEL
LIN {X 0,Y 537.762,Z 265.563,A -85,B 0,C 180,E1 -3881.645,E2 -3881.645} C_VEL
LIN {X 0,Y 537.821,Z 252.096,A -85,B 0,C 180,E1 -3884.761,E2 -3884.761} C_VEL
LIN {X 0,Y 537.859,Z 248.305,A -85,B 0,C 180,E1 -3885.683,E2 -3885.683} C_VEL
LIN {X 0,Y 538,Z 248.278,A -85,B 0,C 180,E1 -3888.271,E2 -3888.271} C_VEL
LIN {X 0,Y 538.002,Z 248.279,A -85,B 0,C 180,E1 -3890.652,E2 -3890.652} C_VEL
LIN {X 0,Y 537.974,Z 248.287,A -85,B 0,C 180,E1 -3893.073,E2 -3893.073} C_VEL
LIN {X 0,Y 537.991,Z 248.283,A -85,B 0,C 180,E1 -3895.66,E2 -3895.66} C_VEL
LIN {X 0,Y 537.971,Z 248.282,A -85,B 0,C 180,E1 -3898.053,E2 -3898.053} C_VEL
LIN {X 0,Y 537.986,Z 248.282,A -85,B 0,C 180,E1 -3900.628,E2 -3900.628} C_VEL
LIN {X 0,Y 538.018,Z 248.282,A -85,B 0,C 180,E1 -3903.278,E2 -3903.278} C_VEL
LIN {X 0,Y 537.965,Z 248.283,A -85,B 0,C 180,E1 -3906.006,E2 -3906.006} C_VEL
LIN {X 0,Y 538.005,Z 248.284,A -85,B 0,C 180,E1 -3908.83,E2 -3908.83} C_VEL
LIN {X 0,Y 537.976,Z 248.281,A -85,B 0,C 180,E1 -3911.872,E2 -3911.872} C_VEL
LIN {X 0,Y 537.989,Z 248.286,A -85,B 0,C 180,E1 -3914.863,E2 -3914.863} C_VEL
LIN {X 0,Y 537.967,Z 248.286,A -85,B 0,C 180,E1 -3917.209,E2 -3917.209} C_VEL
LIN {X 0,Y 538.002,Z 248.282,A -85,B 0,C 180,E1 -3920.418,E2 -3920.418} C_VEL
LIN {X 0,Y 538.012,Z 248.281,A -85,B 0,C 180,E1 -3923.066,E2 -3923.066} C_VEL
LIN {X 0,Y 537.991,Z 248.28,A -85,B 0,C 180,E1 -3925.825,E2 -3925.825} C_VEL
LIN {X 0,Y 537.989,Z 248.286,A -85,B 0,C 180,E1 -3928.497,E2 -3928.497} C_VEL
LIN {X 0,Y 537.979,Z 248.283,A -85,B 0,C 180,E1 -3931.095,E2 -3931.095} C_VEL
LIN {X 0,Y 537.979,Z 248.281,A -85,B 0,C 180,E1 -3933.63,E2 -3933.63} C_VEL
LIN {X 0,Y 537.978,Z 248.286,A -85,B 0,C 180,E1 -3936.128,E2 -3936.128} C_VEL
LIN {X 0,Y 537.992,Z 248.286,A -85,B 0,C 180,E1 -3938.545,E2 -3938.545} C_VEL
LIN {X 0,Y 537.999,Z 248.28,A -85,B 0,C 180,E1 -3940.939,E2 -3940.939} C_VEL
LIN {X 0,Y 537.963,Z 248.283,A -85,B 0,C 180,E1 -3943.297,E2 -3943.297} C_VEL
LIN {X 0,Y 538.031,Z 248.276,A -85,B 0,C 180,E1 -3945.63,E2 -3945.63} C_VEL
LIN {X 0,Y 538.018,Z 248.278,A -85,B 0,C 180,E1 -3948.7,E2 -3948.7} C_VEL
LIN {X 0,Y 538.028,Z 248.279,A -85,B 0,C 180,E1 -3951.739,E2 -3951.739} C_VEL
LIN {X 0,Y 538.117,Z 248.264,A -85,B 0,C 180,E1 -3954.754,E2 -3954.754} C_VEL
LIN {X 0,Y 538.156,Z 248.264,A -85,B 0,C 180,E1 -3957.755,E2 -3957.755} C_VEL
LIN {X 0,Y 538.153,Z 248.266,A -85,B 0,C 180,E1 -3960,E2 -3960} C_VEL
LIN {X 0,Y 538.104,Z 248.265,A -85,B 0,C 180,E1 -3962.995,E2 -3962.995} C_VEL
LIN {X 0,Y 538.075,Z 248.275,A -85,B 0,C 180,E1 -3965.998,E2 -3965.998} C_VEL
LIN {X 0,Y 538.019,Z 248.276,A -85,B 0,C 180,E1 -3969.018,E2 -3969.018} C_VEL
LIN {X 0,Y 538.029,Z 248.278,A -85,B 0,C 180,E1 -3972.064,E2 -3972.064} C_VEL
LIN {X 0,Y 538.029,Z 248.277,A -85,B 0,C 180,E1 -3975.144,E2 -3975.144} C_VEL
LIN {X 0,Y 537.989,Z 248.28,A -85,B 0,C 180,E1 -3978.272,E2 -3978.272} C_VEL
LIN {X 0,Y 537.98,Z 248.281,A -85,B 0,C 180,E1 -3980.654,E2 -3980.654} C_VEL
LIN {X 0,Y 537.969,Z 248.286,A -85,B 0,C 180,E1 -3983.074,E2 -3983.074} C_VEL
LIN {X 0,Y 537.984,Z 248.285,A -85,B 0,C 180,E1 -3985.661,E2 -3985.661} C_VEL
LIN {X 0,Y 537.964,Z 248.283,A -85,B 0,C 180,E1 -3988.054,E2 -3988.054} C_VEL
LIN {X 0,Y 537.981,Z 248.281,A -85,B 0,C 180,E1 -3990.629,E2 -3990.629} C_VEL
LIN {X 0,Y 538.014,Z 248.284,A -85,B 0,C 180,E1 -3993.279,E2 -3993.279} C_VEL
LIN {X 0,Y 537.954,Z 248.284,A -85,B 0,C 180,E1 -3996.008,E2 -3996.008} C_VEL
LIN {X 0,Y 537.994,Z 248.283,A -85,B 0,C 180,E1 -3998.832,E2 -3998.832} C_VEL
LIN {X 0,Y 537.974,Z 248.281,A -85,B 0,C 180,E1 -4001.873,E2 -4001.873} C_VEL
LIN {X 0,Y 537.988,Z 248.285,A -85,B 0,C 180,E1 -4004.864,E2 -4004.864} C_VEL
LIN {X 0,Y 537.965,Z 248.287,A -85,B 0,C 180,E1 -4007.209,E2 -4007.209} C_VEL
LIN {X 0,Y 537.982,Z 248.281,A -85,B 0,C 180,E1 -4010.2,E2 -4010.2} C_VEL
LIN {X 0,Y 537.954,Z 248.288,A -85,B 0,C 180,E1 -4013.062,E2 -4013.062} C_VEL
LIN {X 0,Y 537.983,Z 248.279,A -85,B 0,C 180,E1 -4015.825,E2 -4015.825} C_VEL
LIN {X 0,Y 537.984,Z 248.285,A -85,B 0,C 180,E1 -4018.498,E2 -4018.498} C_VEL
LIN {X 0,Y 537.981,Z 248.283,A -85,B 0,C 180,E1 -4021.096,E2 -4021.096} C_VEL
LIN {X 0,Y 537.972,Z 248.282,A -85,B 0,C 180,E1 -4023.63,E2 -4023.63} C_VEL
LIN {X 0,Y 538.01,Z 248.411,A -85,B 0,C 180,E1 -4026.547,E2 -4026.547} C_VEL
LIN {X 0,Y 538.879,Z 254.407,A -85,B 0,C 180,E1 -4027.575,E2 -4027.575} C_VEL
LIN {X 0,Y 538.593,Z 271.45,A -85,B 0,C 180,E1 -4030.367,E2 -4030.367} C_VEL
LIN {X 0,Y 538.403,Z 287.238,A -85,B 0,C 180,E1 -4032.921,E2 -4032.921} C_VEL
LIN {X 0,Y 538.158,Z 306.61,A -85,B 0,C 180,E1 -4036.02,E2 -4036.02} C_VEL
LIN {X 0,Y 537.935,Z 321.687,A -85,B 0,C 180,E1 -4038.398,E2 -4038.398} C_VEL
LIN {X 0,Y 538.806,Z 330.318,A -85,B 0,C 180,E1 -4038.531,E2 -4038.531} C_VEL
LIN {X 0,Y 538.686,Z 398.527,A -85,B 0,C 180,E1 -4039.452,E2 -4039.452} C_VEL
LIN {X 0,Y 538.522,Z 407.802,A -85,B 0,C 180,E1 -4039.663,E2 -4039.663} C_VEL
LIN {X 0,Y 538.441,Z 416.296,A -85,B 0,C 180,E1 -4039.946,E2 -4039.946} C_VEL
LIN {X 0,Y 538.287,Z 424.826,A -85,B 0,C 180,E1 -4040.323,E2 -4040.323} C_VEL
LIN {X 0,Y 538.21,Z 433.197,A -85,B 0,C 180,E1 -4040.796,E2 -4040.796} C_VEL
LIN {X 0,Y 538.112,Z 441.277,A -85,B 0,C 180,E1 -4041.362,E2 -4041.362} C_VEL
LIN {X 0,Y 537.938,Z 448.97,A -85,B 0,C 180,E1 -4042.021,E2 -4042.021} C_VEL
LIN {X 0,Y 537.852,Z 457.05,A -85,B 0,C 180,E1 -4042.87,E2 -4042.87} C_VEL
LIN {X 0,Y 537.783,Z 463.847,A -85,B 0,C 180,E1 -4043.77,E2 -4043.77} C_VEL
LIN {X 0,Y 537.603,Z 469.699,A -85,B 0,C 180,E1 -4044.75,E2 -4044.75} C_VEL
LIN {X 0,Y 537.624,Z 474.91,A -85,B 0,C 180,E1 -4045.877,E2 -4045.877} C_VEL
LIN {X 0,Y 537.562,Z 478.732,A -85,B 0,C 180,E1 -4047.003,E2 -4047.003} C_VEL
LIN {X 0,Y 537.491,Z 480.488,A -85,B 0,C 180,E1 -4047.752,E2 -4047.752} C_VEL
LIN {X 0,Y 537.45,Z 481.747,A -85,B 0,C 180,E1 -4048.502,E2 -4048.502} C_VEL
LIN {X 0,Y 537.44,Z 482.532,A -85,B 0,C 180,E1 -4049.251,E2 -4049.251} C_VEL
LIN {X 0,Y 537.441,Z 482.829,A -85,B 0,C 180,E1 -4050,E2 -4050} C_VEL
LIN {X 0,Y 537.44,Z 482.531,A -85,B 0,C 180,E1 -4050.75,E2 -4050.75} C_VEL
LIN {X 0,Y 537.45,Z 481.746,A -85,B 0,C 180,E1 -4051.499,E2 -4051.499} C_VEL
LIN {X 0,Y 537.491,Z 480.486,A -85,B 0,C 180,E1 -4052.248,E2 -4052.248} C_VEL
LIN {X 0,Y 537.588,Z 477.568,A -85,B 0,C 180,E1 -4053.373,E2 -4053.373} C_VEL
LIN {X 0,Y 537.624,Z 474.906,A -85,B 0,C 180,E1 -4054.123,E2 -4054.123} C_VEL
LIN {X 0,Y 537.604,Z 469.692,A -85,B 0,C 180,E1 -4055.251,E2 -4055.251} C_VEL
LIN {X 0,Y 537.78,Z 463.865,A -85,B 0,C 180,E1 -4056.227,E2 -4056.227} C_VEL
LIN {X 0,Y 537.853,Z 457.043,A -85,B 0,C 180,E1 -4057.131,E2 -4057.131} C_VEL
LIN {X 0,Y 537.939,Z 448.969,A -85,B 0,C 180,E1 -4057.979,E2 -4057.979} C_VEL
LIN {X 0,Y 538.113,Z 441.271,A -85,B 0,C 180,E1 -4058.639,E2 -4058.639} C_VEL
LIN {X 0,Y 538.211,Z 433.186,A -85,B 0,C 180,E1 -4059.205,E2 -4059.205} C_VEL
LIN {X 0,Y 538.287,Z 424.813,A -85,B 0,C 180,E1 -4059.678,E2 -4059.678} C_VEL
LIN {X 0,Y 538.442,Z 416.279,A -85,B 0,C 180,E1 -4060.054,E2 -4060.054} C_VEL
LIN {X 0,Y 538.526,Z 406.11,A -85,B 0,C 180,E1 -4060.385,E2 -4060.385} C_VEL
LIN {X 0,Y 538.666,Z 394.386,A -85,B 0,C 180,E1 -4060.62,E2 -4060.62} C_VEL
LIN {X 0,Y 538.796,Z 329.109,A -85,B 0,C 180,E1 -4061.485,E2 -4061.485} C_VEL
LIN {X 0,Y 537.942,Z 321.559,A -85,B 0,C 180,E1 -4061.609,E2 -4061.609} C_VEL
LIN {X 0,Y 538.192,Z 302.492,A -85,B 0,C 180,E1 -4064.637,E2 -4064.637} C_VEL
LIN {X 0,Y 538.461,Z 282.124,A -85,B 0,C 180,E1 -4067.903,E2 -4067.903} C_VEL
LIN {X 0,Y 538.707,Z 264.147,A -85,B 0,C 180,E1 -4070.825,E2 -4070.825} C_VEL
LIN {X 0,Y 538.788,Z 253.178,A -85,B 0,C 180,E1 -4072.632,E2 -4072.632} C_VEL
LIN {X 0,Y 538.008,Z 248.284,A -85,B 0,C 180,E1 -4073.48,E2 -4073.48} C_VEL
LIN {X 0,Y 537.974,Z 248.282,A -85,B 0,C 180,E1 -4076.371,E2 -4076.371} C_VEL
LIN {X 0,Y 537.973,Z 248.284,A -85,B 0,C 180,E1 -4078.922,E2 -4078.922} C_VEL
LIN {X 0,Y 537.993,Z 248.279,A -85,B 0,C 180,E1 -4081.884,E2 -4081.884} C_VEL
LIN {X 0,Y 537.987,Z 248.28,A -85,B 0,C 180,E1 -4084.614,E2 -4084.614} C_VEL
LIN {X 0,Y 537.963,Z 248.283,A -85,B 0,C 180,E1 -4087.88,E2 -4087.88} C_VEL
LIN {X 0,Y 537.958,Z 248.287,A -85,B 0,C 180,E1 -4090.784,E2 -4090.784} C_VEL
LIN {X 0,Y 537.997,Z 248.278,A -85,B 0,C 180,E1 -4094.071,E2 -4094.071} C_VEL
LIN {X 0,Y 537.968,Z 248.289,A -85,B 0,C 180,E1 -4097.019,E2 -4097.019} C_VEL
LIN {X 0,Y 537.989,Z 248.283,A -85,B 0,C 180,E1 -4099.26,E2 -4099.26} C_VEL
LIN {X 0,Y 537.967,Z 248.282,A -85,B 0,C 180,E1 -4102.12,E2 -4102.12} C_VEL
LIN {X 0,Y 537.988,Z 248.281,A -85,B 0,C 180,E1 -4105.386,E2 -4105.386} C_VEL
LIN {X 0,Y 537.993,Z 248.28,A -85,B 0,C 180,E1 -4108.116,E2 -4108.116} C_VEL
LIN {X 0,Y 537.984,Z 248.283,A -85,B 0,C 180,E1 -4111.096,E2 -4111.096} C_VEL
LIN {X 0,Y 537.976,Z 248.281,A -85,B 0,C 180,E1 -4113.63,E2 -4113.63} C_VEL
LIN {X 0,Y 537.983,Z 248.283,A -85,B 0,C 180,E1 -4116.128,E2 -4116.128} C_VEL
LIN {X 0,Y 537.988,Z 248.287,A -85,B 0,C 180,E1 -4118.545,E2 -4118.545} C_VEL
LIN {X 0,Y 537.956,Z 248.286,A -85,B 0,C 180,E1 -4120.937,E2 -4120.937} C_VEL
LIN {X 0,Y 537.968,Z 248.282,A -85,B 0,C 180,E1 -4123.297,E2 -4123.297} C_VEL
LIN {X 0,Y 538.021,Z 248.276,A -85,B 0,C 180,E1 -4125.63,E2 -4125.63} C_VEL
LIN {X 0,Y 538.023,Z 248.279,A -85,B 0,C 180,E1 -4128.7,E2 -4128.7} C_VEL
LIN {X 0,Y 538.034,Z 248.276,A -85,B 0,C 180,E1 -4131.739,E2 -4131.739} C_VEL
LIN {X 0,Y 538.119,Z 248.265,A -85,B 0,C 180,E1 -4134.755,E2 -4134.755} C_VEL
LIN {X 0,Y 538.161,Z 248.262,A -85,B 0,C 180,E1 -4137.755,E2 -4137.755} C_VEL
LIN {X 0,Y 538.159,Z 248.266,A -85,B 0,C 180,E1 -4140,E2 -4140} C_VEL
LIN {X 0,Y 538.109,Z 248.265,A -85,B 0,C 180,E1 -4142.995,E2 -4142.995} C_VEL
LIN {X 0,Y 538.08,Z 248.275,A -85,B 0,C 180,E1 -4145.998,E2 -4145.998} C_VEL
LIN {X 0,Y 538.025,Z 248.275,A -85,B 0,C 180,E1 -4149.018,E2 -4149.018} C_VEL
LIN {X 0,Y 538.036,Z 248.28,A -85,B 0,C 180,E1 -4152.064,E2 -4152.064} C_VEL
LIN {X 0,Y 538.037,Z 248.275,A -85,B 0,C 180,E1 -4155.144,E2 -4155.144} C_VEL
LIN {X 0,Y 537.996,Z 248.281,A -85,B 0,C 180,E1 -4158.272,E2 -4158.272} C_VEL
LIN {X 0,Y 537.987,Z 248.28,A -85,B 0,C 180,E1 -4160.654,E2 -4160.654} C_VEL
LIN {X 0,Y 537.976,Z 248.283,A -85,B 0,C 180,E1 -4163.074,E2 -4163.074} C_VEL
LIN {X 0,Y 537.995,Z 248.285,A -85,B 0,C 180,E1 -4165.661,E2 -4165.661} C_VEL
LIN {X 0,Y 537.972,Z 248.284,A -85,B 0,C 180,E1 -4168.054,E2 -4168.054} C_VEL
LIN {X 0,Y 537.993,Z 248.279,A -85,B 0,C 180,E1 -4170.629,E2 -4170.629} C_VEL
LIN {X 0,Y 538.021,Z 248.282,A -85,B 0,C 180,E1 -4173.278,E2 -4173.278} C_VEL
LIN {X 0,Y 537.97,Z 248.283,A -85,B 0,C 180,E1 -4176.007,E2 -4176.007} C_VEL
LIN {X 0,Y 538.007,Z 248.28,A -85,B 0,C 180,E1 -4178.831,E2 -4178.831} C_VEL
LIN {X 0,Y 537.98,Z 248.281,A -85,B 0,C 180,E1 -4180.22,E2 -4180.22} C_VEL
LIN {X 0,Y 537.314,Z 248.368,A -85,B 0,C 180,E1 -4180.845,E2 -4180.845} C_VEL
LIN {X 0,Y 534.462,Z 248.728,A -85,B 0,C 180,E1 -4181.86,E2 -4181.86} C_VEL
LIN {X 0,Y 532.05,Z 249.03,A -85,B 0,C 180,E1 -4182.677,E2 -4182.677} C_VEL
LIN {X 0,Y 531.012,Z 249.156,A -85,B 0,C 180,E1 -4183.308,E2 -4183.308} C_VEL
LIN {X 0,Y 530.927,Z 249.164,A -85,B 0,C 180,E1 -4183.521,E2 -4183.521} C_VEL
LIN {X 0,Y 530.966,Z 249.158,A -85,B 0,C 180,E1 -4185.623,E2 -4185.623} C_VEL
LIN {X 0,Y 530.936,Z 249.164,A -85,B 0,C 180,E1 -4188.983,E2 -4188.983} C_VEL
LIN {X 0,Y 530.952,Z 249.159,A -85,B 0,C 180,E1 -4191.529,E2 -4191.529} C_VEL
LIN {X 0,Y 530.948,Z 249.158,A -85,B 0,C 180,E1 -4194.379,E2 -4194.379} C_VEL
LIN {X 0,Y 530.966,Z 249.161,A -85,B 0,C 180,E1 -4197.133,E2 -4197.133} C_VEL
LIN {X 0,Y 530.936,Z 249.158,A -85,B 0,C 180,E1 -4199.801,E2 -4199.801} C_VEL
LIN {X 0,Y 530.964,Z 249.159,A -85,B 0,C 180,E1 -4202.478,E2 -4202.478} C_VEL
LIN {X 0,Y 530.949,Z 249.164,A -85,B 0,C 180,E1 -4204.939,E2 -4204.939} C_VEL
LIN {X 0,Y 530.973,Z 249.154,A -85,B 0,C 180,E1 -4207.9,E2 -4207.9} C_VEL
LIN {X 0,Y 530.971,Z 249.163,A -85,B 0,C 180,E1 -4210.676,E2 -4210.676} C_VEL
LIN {X 0,Y 530.935,Z 249.162,A -85,B 0,C 180,E1 -4213.069,E2 -4213.069} C_VEL
LIN {X 0,Y 530.826,Z 249.245,A -85,B 0,C 180,E1 -4214.497,E2 -4214.497} C_VEL
LIN {X 0,Y 530.734,Z 263.433,A -85,B 0,C 180,E1 -4217.768,E2 -4217.768} C_VEL
LIN {X 0,Y 530.725,Z 265.826,A -85,B 0,C 180,E1 -4218.309,E2 -4218.309} C_VEL
LIN {X 0,Y 531.94,Z 275.088,A -85,B 0,C 180,E1 -4218.463,E2 -4218.463} C_VEL
LIN {X 0,Y 531.674,Z 340.57,A -85,B 0,C 180,E1 -4219.359,E2 -4219.359} C_VEL
LIN {X 0,Y 531.606,Z 348.944,A -85,B 0,C 180,E1 -4219.55,E2 -4219.55} C_VEL
LIN {X 0,Y 531.503,Z 358.202,A -85,B 0,C 180,E1 -4219.861,E2 -4219.861} C_VEL
LIN {X 0,Y 531.407,Z 365.731,A -85,B 0,C 180,E1 -4220.196,E2 -4220.196} C_VEL
LIN {X 0,Y 531.293,Z 374.207,A -85,B 0,C 180,E1 -4220.674,E2 -4220.674} C_VEL
LIN {X 0,Y 531.189,Z 382.337,A -85,B 0,C 180,E1 -4221.248,E2 -4221.248} C_VEL
LIN {X 0,Y 531.03,Z 390.051,A -85,B 0,C 180,E1 -4221.916,E2 -4221.916} C_VEL
LIN {X 0,Y 530.903,Z 396.416,A -85,B 0,C 180,E1 -4222.584,E2 -4222.584} C_VEL
LIN {X 0,Y 530.803,Z 403.563,A -85,B 0,C 180,E1 -4223.495,E2 -4223.495} C_VEL
LIN {X 0,Y 530.553,Z 410.744,A -85,B 0,C 180,E1 -4224.679,E2 -4224.679} C_VEL
LIN {X 0,Y 530.623,Z 414.401,A -85,B 0,C 180,E1 -4225.442,E2 -4225.442} C_VEL
LIN {X 0,Y 530.527,Z 417.391,A -85,B 0,C 180,E1 -4226.202,E2 -4226.202} C_VEL
LIN {X 0,Y 530.527,Z 419.704,A -85,B 0,C 180,E1 -4226.962,E2 -4226.962} C_VEL
LIN {X 0,Y 530.414,Z 421.476,A -85,B 0,C 180,E1 -4227.722,E2 -4227.722} C_VEL
LIN {X 0,Y 530.371,Z 422.753,A -85,B 0,C 180,E1 -4228.481,E2 -4228.481} C_VEL
LIN {X 0,Y 530.362,Z 423.562,A -85,B 0,C 180,E1 -4229.24,E2 -4229.24} C_VEL
LIN {X 0,Y 530.363,Z 423.87,A -85,B 0,C 180,E1 -4230,E2 -4230} C_VEL
LIN {X 0,Y 530.363,Z 423.6,A -85,B 0,C 180,E1 -4230.759,E2 -4230.759} C_VEL
LIN {X 0,Y 530.371,Z 422.868,A -85,B 0,C 180,E1 -4231.518,E2 -4231.518} C_VEL
LIN {X 0,Y 530.414,Z 421.668,A -85,B 0,C 180,E1 -4232.278,E2 -4232.278} C_VEL
LIN {X 0,Y 530.549,Z 418.836,A -85,B 0,C 180,E1 -4233.417,E2 -4233.417} C_VEL
LIN {X 0,Y 530.558,Z 416.266,A -85,B 0,C 180,E1 -4234.178,E2 -4234.178} C_VEL
LIN {X 0,Y 530.543,Z 411.199,A -85,B 0,C 180,E1 -4235.32,E2 -4235.32} C_VEL
LIN {X 0,Y 530.789,Z 405.644,A -85,B 0,C 180,E1 -4236.285,E2 -4236.285} C_VEL
LIN {X 0,Y 530.854,Z 398.883,A -85,B 0,C 180,E1 -4237.225,E2 -4237.225} C_VEL
LIN {X 0,Y 531.018,Z 391.007,A -85,B 0,C 180,E1 -4238.083,E2 -4238.083} C_VEL
LIN {X 0,Y 531.194,Z 383.49,A -85,B 0,C 180,E1 -4238.751,E2 -4238.751} C_VEL
LIN {X 0,Y 531.297,Z 375.617,A -85,B 0,C 180,E1 -4239.325,E2 -4239.325} C_VEL
LIN {X 0,Y 531.406,Z 367.491,A -85,B 0,C 180,E1 -4239.803,E2 -4239.803} C_VEL
LIN {X 0,Y 531.526,Z 359.267,A -85,B 0,C 180,E1 -4240.186,E2 -4240.186} C_VEL
LIN {X 0,Y 531.575,Z 350.412,A -85,B 0,C 180,E1 -4240.498,E2 -4240.498} C_VEL
LIN {X 0,Y 531.755,Z 341.562,A -85,B 0,C 180,E1 -4240.711,E2 -4240.711} C_VEL
LIN {X 0,Y 531.897,Z 281.808,A -85,B 0,C 180,E1 -4241.537,E2 -4241.537} C_VEL
LIN {X 0,Y 531.739,Z 272.205,A -85,B 0,C 180,E1 -4241.671,E2 -4241.671} C_VEL
LIN {X 0,Y 530.737,Z 265.755,A -85,B 0,C 180,E1 -4241.8,E2 -4241.8} C_VEL
LIN {X 0,Y 530.774,Z 251.613,A -85,B 0,C 180,E1 -4245.042,E2 -4245.042} C_VEL
LIN {X 0,Y 530.828,Z 249.181,A -85,B 0,C 180,E1 -4245.649,E2 -4245.649} C_VEL
LIN {X 0,Y 530.971,Z 249.159,A -85,B 0,C 180,E1 -4247.723,E2 -4247.723} C_VEL
LIN {X 0,Y 531.008,Z 249.15,A -85,B 0,C 180,E1 -4250.127,E2 -4250.127} C_VEL
LIN {X 0,Y 530.915,Z 249.161,A -85,B 0,C 180,E1 -4252.574,E2 -4252.574} C_VEL
LIN {X 0,Y 530.945,Z 249.163,A -85,B 0,C 180,E1 -4255.06,E2 -4255.06} C_VEL
LIN {X 0,Y 530.951,Z 249.16,A -85,B 0,C 180,E1 -4257.598,E2 -4257.598} C_VEL
LIN {X 0,Y 530.94,Z 249.16,A -85,B 0,C 180,E1 -4260.639,E2 -4260.639} C_VEL
LIN {X 0,Y 530.958,Z 249.159,A -85,B 0,C 180,E1 -4263.499,E2 -4263.499} C_VEL
LIN {X 0,Y 530.94,Z 249.16,A -85,B 0,C 180,E1 -4266.559,E2 -4266.559} C_VEL
LIN {X 0,Y 530.963,Z 249.158,A -85,B 0,C 180,E1 -4269.445,E2 -4269.445} C_VEL
LIN {X 0,Y 530.911,Z 249.164,A -85,B 0,C 180,E1 -4272.463,E2 -4272.463} C_VEL
LIN {X 0,Y 530.959,Z 249.157,A -85,B 0,C 180,E1 -4275.45,E2 -4275.45} C_VEL
LIN {X 0,Y 530.946,Z 249.163,A -85,B 0,C 180,E1 -4278.56,E2 -4278.56} C_VEL
LIN {X 0,Y 530.944,Z 249.158,A -85,B 0,C 180,E1 -4281.528,E2 -4281.528} C_VEL
LIN {X 0,Y 530.93,Z 249.164,A -85,B 0,C 180,E1 -4284.378,E2 -4284.378} C_VEL
LIN {X 0,Y 530.96,Z 249.158,A -85,B 0,C 180,E1 -4287.133,E2 -4287.133} C_VEL
LIN {X 0,Y 530.927,Z 249.16,A -85,B 0,C 180,E1 -4289.8,E2 -4289.8} C_VEL
LIN {X 0,Y 530.949,Z 249.163,A -85,B 0,C 180,E1 -4292.48,E2 -4292.48} C_VEL
LIN {X 0,Y 530.943,Z 249.16,A -85,B 0,C 180,E1 -4294.939,E2 -4294.939} C_VEL
LIN {X 0,Y 530.945,Z 249.163,A -85,B 0,C 180,E1 -4298.245,E2 -4298.245} C_VEL
LIN {X 0,Y 530.956,Z 249.16,A -85,B 0,C 180,E1 -4300.676,E2 -4300.676} C_VEL
LIN {X 0,Y 530.931,Z 249.16,A -85,B 0,C 180,E1 -4303.069,E2 -4303.069} C_VEL
LIN {X 0,Y 530.992,Z 249.152,A -85,B 0,C 180,E1 -4305.435,E2 -4305.435} C_VEL
LIN {X 0,Y 530.98,Z 249.157,A -85,B 0,C 180,E1 -4308.548,E2 -4308.548} C_VEL
LIN {X 0,Y 530.976,Z 249.156,A -85,B 0,C 180,E1 -4311.628,E2 -4311.628} C_VEL
LIN {X 0,Y 531.079,Z 249.142,A -85,B 0,C 180,E1 -4314.685,E2 -4314.685} C_VEL
LIN {X 0,Y 531.128,Z 249.14,A -85,B 0,C 180,E1 -4317.725,E2 -4317.725} C_VEL
LIN {X 0,Y 531.122,Z 249.142,A -85,B 0,C 180,E1 -4320,E2 -4320} C_VEL
LIN {X 0,Y 531.127,Z 249.138,A -85,B 0,C 180,E1 -4322.275,E2 -4322.275} C_VEL
LIN {X 0,Y 531.076,Z 249.143,A -85,B 0,C 180,E1 -4325.315,E2 -4325.315} C_VEL
LIN {X 0,Y 530.976,Z 249.155,A -85,B 0,C 180,E1 -4328.372,E2 -4328.372} C_VEL
LIN {X 0,Y 531.005,Z 249.156,A -85,B 0,C 180,E1 -4331.65,E2 -4331.65} C_VEL
LIN {X 0,Y 531.012,Z 249.15,A -85,B 0,C 180,E1 -4334.95,E2 -4334.95} C_VEL
LIN {X 0,Y 530.964,Z 249.161,A -85,B 0,C 180,E1 -4337.724,E2 -4337.724} C_VEL
LIN {X 0,Y 530.965,Z 249.156,A -85,B 0,C 180,E1 -4340.129,E2 -4340.129} C_VEL
LIN {X 0,Y 530.91,Z 249.161,A -85,B 0,C 180,E1 -4342.575,E2 -4342.575} C_VEL
LIN {X 0,Y 530.937,Z 249.162,A -85,B 0,C 180,E1 -4345.061,E2 -4345.061} C_VEL
LIN {X 0,Y 530.944,Z 249.162,A -85,B 0,C 180,E1 -4347.599,E2 -4347.599} C_VEL
LIN {X 0,Y 530.935,Z 249.159,A -85,B 0,C 180,E1 -4350.639,E2 -4350.639} C_VEL
LIN {X 0,Y 530.955,Z 249.16,A -85,B 0,C 180,E1 -4353.5,E2 -4353.5} C_VEL
LIN {X 0,Y 530.902,Z 249.162,A -85,B 0,C 180,E1 -4356.148,E2 -4356.148} C_VEL
LIN {X 0,Y 530.949,Z 249.159,A -85,B 0,C 180,E1 -4358.652,E2 -4358.652} C_VEL
LIN {X 0,Y 530.945,Z 249.16,A -85,B 0,C 180,E1 -4361.44,E2 -4361.44} C_VEL
LIN {X 0,Y 530.958,Z 249.158,A -85,B 0,C 180,E1 -4364.55,E2 -4364.55} C_VEL
LIN {X 0,Y 530.908,Z 249.162,A -85,B 0,C 180,E1 -4367.537,E2 -4367.537} C_VEL
LIN {X 0,Y 530.948,Z 249.16,A -85,B 0,C 180,E1 -4370.554,E2 -4370.554} C_VEL
LIN {X 0,Y 530.902,Z 249.163,A -85,B 0,C 180,E1 -4373.438,E2 -4373.438} C_VEL
LIN {X 0,Y 530.927,Z 249.16,A -85,B 0,C 180,E1 -4376.224,E2 -4376.224} C_VEL
LIN {X 0,Y 530.931,Z 249.163,A -85,B 0,C 180,E1 -4378.92,E2 -4378.92} C_VEL
LIN {X 0,Y 530.926,Z 249.159,A -85,B 0,C 180,E1 -4381.541,E2 -4381.541} C_VEL
LIN {X 0,Y 530.923,Z 249.164,A -85,B 0,C 180,E1 -4384.176,E2 -4384.176} C_VEL
LIN {X 0,Y 530.992,Z 249.258,A -85,B 0,C 180,E1 -4386.425,E2 -4386.425} C_VEL
LIN {X 0,Y 531.884,Z 255.256,A -85,B 0,C 180,E1 -4387.469,E2 -4387.469} C_VEL
LIN {X 0,Y 531.606,Z 271.075,A -85,B 0,C 180,E1 -4390.098,E2 -4390.098} C_VEL
LIN {X 0,Y 531.367,Z 285.641,A -85,B 0,C 180,E1 -4392.489,E2 -4392.489} C_VEL
LIN {X 0,Y 531.124,Z 303.801,A -85,B 0,C 180,E1 -4395.439,E2 -4395.439} C_VEL
LIN {X 0,Y 530.888,Z 321.14,A -85,B 0,C 180,E1 -4398.231,E2 -4398.231} C_VEL
LIN {X 0,Y 531.856,Z 330.56,A -85,B 0,C 180,E1 -4398.388,E2 -4398.388} C_VEL
LIN {X 0,Y 531.684,Z 398.133,A -85,B 0,C 180,E1 -4399.312,E2 -4399.312} C_VEL
LIN {X 0,Y 531.543,Z 407.411,A -85,B 0,C 180,E1 -4399.526,E2 -4399.526} C_VEL
LIN {X 0,Y 531.448,Z 415.903,A -85,B 0,C 180,E1 -4399.813,E2 -4399.813} C_VEL
LIN {X 0,Y 531.284,Z 424.434,A -85,B 0,C 180,E1 -4400.194,E2 -4400.194} C_VEL
LIN {X 0,Y 531.186,Z 432.804,A -85,B 0,C 180,E1 -4400.673,E2 -4400.673} C_VEL
LIN {X 0,Y 531.075,Z 440.884,A -85,B 0,C 180,E1 -4401.247,E2 -4401.247} C_VEL
LIN {X 0,Y 530.895,Z 448.578,A -85,B 0,C 180,E1 -4401.915,E2 -4401.915} C_VEL
LIN {X 0,Y 530.771,Z 456.656,A -85,B 0,C 180,E1 -4402.774,E2 -4402.774} C_VEL
LIN {X 0,Y 530.684,Z 463.787,A -85,B 0,C 180,E1 -4403.74,E2 -4403.74} C_VEL
LIN {X 0,Y 530.541,Z 469.308,A -85,B 0,C 180,E1 -4404.68,E2 -4404.68} C_VEL
LIN {X 0,Y 530.546,Z 474.518,A -85,B 0,C 180,E1 -4405.822,E2 -4405.822} C_VEL
LIN {X 0,Y 530.469,Z 478.34,A -85,B 0,C 180,E1 -4406.963,E2 -4406.963} C_VEL
LIN {X 0,Y 530.412,Z 480.097,A -85,B 0,C 180,E1 -4407.722,E2 -4407.722} C_VEL
LIN {X 0,Y 530.36,Z 481.356,A -85,B 0,C 180,E1 -4408.482,E2 -4408.482} C_VEL
LIN {X 0,Y 530.35,Z 482.14,A -85,B 0,C 180,E1 -4409.241,E2 -4409.241} C_VEL
LIN {X 0,Y 530.352,Z 482.438,A -85,B 0,C 180,E1 -4410,E2 -4410} C_VEL
LIN {X 0,Y 530.35,Z 482.14,A -85,B 0,C 180,E1 -4410.76,E2 -4410.76} C_VEL
LIN {X 0,Y 530.36,Z 481.354,A -85,B 0,C 180,E1 -4411.519,E2 -4411.519} C_VEL
LIN {X 0,Y 530.412,Z 480.095,A -85,B 0,C 180,E1 -4412.279,E2 -4412.279} C_VEL
LIN {X 0,Y 530.494,Z 477.176,A -85,B 0,C 180,E1 -4413.418,E2 -4413.418} C_VEL
LIN {X 0,Y 530.546,Z 474.515,A -85,B 0,C 180,E1 -4414.178,E2 -4414.178} C_VEL
LIN {X 0,Y 530.542,Z 469.301,A -85,B 0,C 180,E1 -4415.321,E2 -4415.321} C_VEL
LIN {X 0,Y 530.67,Z 462.673,A -85,B 0,C 180,E1 -4416.431,E2 -4416.431} C_VEL
LIN {X 0,Y 530.785,Z 454.941,A -85,B 0,C 180,E1 -4417.418,E2 -4417.418} C_VEL
LIN {X 0,Y 530.904,Z 447.549,A -85,B 0,C 180,E1 -4418.182,E2 -4418.182} C_VEL
LIN {X 0,Y 531.065,Z 439.639,A -85,B 0,C 180,E1 -4418.85,E2 -4418.85} C_VEL
LIN {X 0,Y 531.196,Z 431.285,A -85,B 0,C 180,E1 -4419.424,E2 -4419.424} C_VEL
LIN {X 0,Y 531.362,Z 420.626,A -85,B 0,C 180,E1 -4419.997,E2 -4419.997} C_VEL
LIN {X 0,Y 531.53,Z 409.053,A -85,B 0,C 180,E1 -4420.427,E2 -4420.427} C_VEL
LIN {X 0,Y 531.622,Z 399.387,A -85,B 0,C 180,E1 -4420.666,E2 -4420.666} C_VEL
LIN {X 0,Y 531.864,Z 330.264,A -85,B 0,C 180,E1 -4421.616,E2 -4421.616} C_VEL
LIN {X 0,Y 530.894,Z 321.115,A -85,B 0,C 180,E1 -4421.773,E2 -4421.773} C_VEL
LIN {X 0,Y 531.136,Z 301.837,A -85,B 0,C 180,E1 -4424.878,E2 -4424.878} C_VEL
LIN {X 0,Y 531.513,Z 280.909,A -85,B 0,C 180,E1 -4428.283,E2 -4428.283} C_VEL
LIN {X 0,Y 531.764,Z 261.34,A -85,B 0,C 180,E1 -4431.516,E2 -4431.516} C_VEL
LIN {X 0,Y 531.777,Z 254.028,A -85,B 0,C 180,E1 -4432.742,E2 -4432.742} C_VEL
LIN {X 0,Y 530.96,Z 249.162,A -85,B 0,C 180,E1 -4433.623,E2 -4433.623} C_VEL
LIN {X 0,Y 530.94,Z 249.159,A -85,B 0,C 180,E1 -4436.747,E2 -4436.747} C_VEL
LIN {X 0,Y 530.914,Z 249.169,A -85,B 0,C 180,E1 -4439.327,E2 -4439.327} C_VEL
LIN {X 0,Y 530.949,Z 249.156,A -85,B 0,C 180,E1 -4442.097,E2 -4442.097} C_VEL
LIN {X 0,Y 530.949,Z 249.159,A -85,B 0,C 180,E1 -4444.848,E2 -4444.848} C_VEL
LIN {X 0,Y 530.904,Z 249.165,A -85,B 0,C 180,E1 -4447.513,E2 -4447.513} C_VEL
LIN {X 0,Y 530.913,Z 249.161,A -85,B 0,C 180,E1 -4450.439,E2 -4450.439} C_VEL
LIN {X 0,Y 530.92,Z 249.162,A -85,B 0,C 180,E1 -4453.5,E2 -4453.5} C_VEL
LIN {X 0,Y 530.964,Z 249.155,A -85,B 0,C 180,E1 -4455.624,E2 -4455.624} C_VEL
LIN {X 0,Y 530.926,Z 249.166,A -85,B 0,C 180,E1 -4458.984,E2 -4458.984} C_VEL
LIN {X 0,Y 530.928,Z 249.16,A -85,B 0,C 180,E1 -4461.527,E2 -4461.527} C_VEL
LIN {X 0,Y 530.924,Z 249.162,A -85,B 0,C 180,E1 -4464.378,E2 -4464.378} C_VEL
LIN {X 0,Y 530.944,Z 249.161,A -85,B 0,C 180,E1 -4467.132,E2 -4467.132} C_VEL
LIN {X 0,Y 530.928,Z 249.159,A -85,B 0,C 180,E1 -4469.801,E2 -4469.801} C_VEL
LIN {X 0,Y 530.954,Z 249.162,A -85,B 0,C 180,E1 -4472.48,E2 -4472.48} C_VEL
LIN {X 0,Y 530.933,Z 249.163,A -85,B 0,C 180,E1 -4474.939,E2 -4474.939} C_VEL
LIN {X 0,Y 530.958,Z 249.156,A -85,B 0,C 180,E1 -4477.904,E2 -4477.904} C_VEL
LIN {X 0,Y 530.915,Z 249.166,A -85,B 0,C 180,E1 -4480.674,E2 -4480.674} C_VEL
LIN {X 0,Y 530.931,Z 249.16,A -85,B 0,C 180,E1 -4483.069,E2 -4483.069} C_VEL
LIN {X 0,Y 530.974,Z 249.153,A -85,B 0,C 180,E1 -4485.435,E2 -4485.435} C_VEL
LIN {X 0,Y 530.986,Z 249.157,A -85,B 0,C 180,E1 -4488.549,E2 -4488.549} C_VEL
LIN {X 0,Y 530.982,Z 249.154,A -85,B 0,C 180,E1 -4491.628,E2 -4491.628} C_VEL
LIN {X 0,Y 531.081,Z 249.143,A -85,B 0,C 180,E1 -4494.685,E2 -4494.685} C_VEL
LIN {X 0,Y 531.132,Z 249.137,A -85,B 0,C 180,E1 -4497.725,E2 -4497.725} C_VEL
LIN {X 0,Y 531.128,Z 249.141,A -85,B 0,C 180,E1 -4500,E2 -4500} C_VEL
LIN {X 0,Y 531.133,Z 249.139,A -85,B 0,C 180,E1 -4502.275,E2 -4502.275} C_VEL
LIN {X 0,Y 531.081,Z 249.141,A -85,B 0,C 180,E1 -4505.315,E2 -4505.315} C_VEL
LIN {X 0,Y 530.983,Z 249.156,A -85,B 0,C 180,E1 -4508.372,E2 -4508.372} C_VEL
LIN {X 0,Y 531.012,Z 249.155,A -85,B 0,C 180,E1 -4511.65,E2 -4511.65} C_VEL
LIN {X 0,Y 531.02,Z 249.148,A -85,B 0,C 180,E1 -4514.95,E2 -4514.95} C_VEL
LIN {X 0,Y 530.972,Z 249.16,A -85,B 0,C 180,E1 -4517.724,E2 -4517.724} C_VEL
LIN {X 0,Y 530.972,Z 249.157,A -85,B 0,C 180,E1 -4520.129,E2 -4520.129} C_VEL
LIN {X 0,Y 530.917,Z 249.161,A -85,B 0,C 180,E1 -4522.575,E2 -4522.575} C_VEL
LIN {X 0,Y 530.949,Z 249.159,A -85,B 0,C 180,E1 -4525.061,E2 -4525.061} C_VEL
LIN {X 0,Y 530.951,Z 249.162,A -85,B 0,C 180,E1 -4527.599,E2 -4527.599} C_VEL
LIN {X 0,Y 530.947,Z 249.157,A -85,B 0,C 180,E1 -4530.64,E2 -4530.64} C_VEL
LIN {X 0,Y 530.962,Z 249.161,A -85,B 0,C 180,E1 -4533.499,E2 -4533.499} C_VEL
LIN {X 0,Y 530.944,Z 249.158,A -85,B 0,C 180,E1 -4536.56,E2 -4536.56} C_VEL
LIN {X 0,Y 530.965,Z 249.161,A -85,B 0,C 180,E1 -4539.445,E2 -4539.445} C_VEL
LIN {X 0,Y 530.915,Z 249.162,A -85,B 0,C 180,E1 -4542.463,E2 -4542.463} C_VEL
LIN {X 0,Y 530.927,Z 249.164,A -85,B 0,C 180,E1 -4543.521,E2 -4543.521} C_VEL
LIN {X 0,Y 530.262,Z 249.243,A -85,B 0,C 180,E1 -4544.155,E2 -4544.155} C_VEL
LIN {X 0,Y 527.423,Z 249.602,A -85,B 0,C 180,E1 -4545.184,E2 -4545.184} C_VEL
LIN {X 0,Y 525.017,Z 249.903,A -85,B 0,C 180,E1 -4546.012,E2 -4546.012} C_VEL
LIN {X 0,Y 523.971,Z 250.032,A -85,B 0,C 180,E1 -4546.652,E2 -4546.652} C_VEL
LIN {X 0,Y 523.879,Z 250.042,A -85,B 0,C 180,E1 -4546.868,E2 -4546.868} C_VEL
LIN {X 0,Y 523.914,Z 250.034,A -85,B 0,C 180,E1 -4549.917,E2 -4549.917} C_VEL
LIN {X 0,Y 523.905,Z 250.04,A -85,B 0,C 180,E1 -4552.867,E2 -4552.867} C_VEL
LIN {X 0,Y 523.913,Z 250.034,A -85,B 0,C 180,E1 -4555.708,E2 -4555.708} C_VEL
LIN {X 0,Y 523.909,Z 250.037,A -85,B 0,C 180,E1 -4558.455,E2 -4558.455} C_VEL
LIN {X 0,Y 523.902,Z 250.04,A -85,B 0,C 180,E1 -4561.123,E2 -4561.123} C_VEL
LIN {X 0,Y 523.913,Z 250.034,A -85,B 0,C 180,E1 -4563.997,E2 -4563.997} C_VEL
LIN {X 0,Y 523.907,Z 250.037,A -85,B 0,C 180,E1 -4566.269,E2 -4566.269} C_VEL
LIN {X 0,Y 523.936,Z 250.037,A -85,B 0,C 180,E1 -4568.766,E2 -4568.766} C_VEL
LIN {X 0,Y 523.929,Z 250.033,A -85,B 0,C 180,E1 -4571.22,E2 -4571.22} C_VEL
LIN {X 0,Y 523.87,Z 250.04,A -85,B 0,C 180,E1 -4573.636,E2 -4573.636} C_VEL
LIN {X 0,Y 523.766,Z 250.122,A -85,B 0,C 180,E1 -4574.526,E2 -4574.526} C_VEL
LIN {X 0,Y 523.683,Z 263.561,A -85,B 0,C 180,E1 -4577.6,E2 -4577.6} C_VEL
LIN {X 0,Y 523.711,Z 265.95,A -85,B 0,C 180,E1 -4578.134,E2 -4578.134} C_VEL
LIN {X 0,Y 525.012,Z 275.523,A -85,B 0,C 180,E1 -4578.308,E2 -4578.308} C_VEL
LIN {X 0,Y 524.719,Z 340.993,A -85,B 0,C 180,E1 -4579.216,E2 -4579.216} C_VEL
LIN {X 0,Y 524.65,Z 349.356,A -85,B 0,C 180,E1 -4579.41,E2 -4579.41} C_VEL
LIN {X 0,Y 524.538,Z 358.608,A -85,B 0,C 180,E1 -4579.725,E2 -4579.725} C_VEL
LIN {X 0,Y 524.44,Z 366.134,A -85,B 0,C 180,E1 -4580.064,E2 -4580.064} C_VEL
LIN {X 0,Y 524.306,Z 374.607,A -85,B 0,C 180,E1 -4580.549,E2 -4580.549} C_VEL
LIN {X 0,Y 524.203,Z 382.735,A -85,B 0,C 180,E1 -4581.13,E2 -4581.13} C_VEL
LIN {X 0,Y 524.036,Z 390.448,A -85,B 0,C 180,E1 -4581.807,E2 -4581.807} C_VEL
LIN {X 0,Y 523.889,Z 396.812,A -85,B 0,C 180,E1 -4582.484,E2 -4582.484} C_VEL
LIN {X 0,Y 523.759,Z 404.393,A -85,B 0,C 180,E1 -4583.467,E2 -4583.467} C_VEL
LIN {X 0,Y 523.493,Z 411.139,A -85,B 0,C 180,E1 -4584.607,E2 -4584.607} C_VEL
LIN {X 0,Y 523.567,Z 414.794,A -85,B 0,C 180,E1 -4585.38,E2 -4585.38} C_VEL
LIN {X 0,Y 523.457,Z 417.784,A -85,B 0,C 180,E1 -4586.15,E2 -4586.15} C_VEL
LIN {X 0,Y 523.464,Z 420.096,A -85,B 0,C 180,E1 -4586.921,E2 -4586.921} C_VEL
LIN {X 0,Y 523.34,Z 421.868,A -85,B 0,C 180,E1 -4587.691,E2 -4587.691} C_VEL
LIN {X 0,Y 523.284,Z 423.145,A -85,B 0,C 180,E1 -4588.46,E2 -4588.46} C_VEL
LIN {X 0,Y 523.274,Z 423.954,A -85,B 0,C 180,E1 -4589.23,E2 -4589.23} C_VEL
LIN {X 0,Y 523.275,Z 424.261,A -85,B 0,C 180,E1 -4590,E2 -4590} C_VEL
LIN {X 0,Y 523.275,Z 423.991,A -85,B 0,C 180,E1 -4590.769,E2 -4590.769} C_VEL
LIN {X 0,Y 523.284,Z 423.258,A -85,B 0,C 180,E1 -4591.539,E2 -4591.539} C_VEL
LIN {X 0,Y 523.34,Z 422.058,A -85,B 0,C 180,E1 -4592.309,E2 -4592.309} C_VEL
LIN {X 0,Y 523.482,Z 419.225,A -85,B 0,C 180,E1 -4593.463,E2 -4593.463} C_VEL
LIN {X 0,Y 523.494,Z 416.655,A -85,B 0,C 180,E1 -4594.234,E2 -4594.234} C_VEL
LIN {X 0,Y 523.486,Z 411.587,A -85,B 0,C 180,E1 -4595.392,E2 -4595.392} C_VEL
LIN {X 0,Y 523.739,Z 406.207,A -85,B 0,C 180,E1 -4596.341,E2 -4596.341} C_VEL
LIN {X 0,Y 523.819,Z 399.269,A -85,B 0,C 180,E1 -4597.322,E2 -4597.322} C_VEL
LIN {X 0,Y 524.015,Z 390.377,A -85,B 0,C 180,E1 -4598.289,E2 -4598.289} C_VEL
LIN {X 0,Y 524.198,Z 382.652,A -85,B 0,C 180,E1 -4598.966,E2 -4598.966} C_VEL
LIN {X 0,Y 524.283,Z 374.508,A -85,B 0,C 180,E1 -4599.548,E2 -4599.548} C_VEL
LIN {X 0,Y 524.453,Z 366.004,A -85,B 0,C 180,E1 -4600.032,E2 -4600.032} C_VEL
LIN {X 0,Y 524.602,Z 354.776,A -85,B 0,C 180,E1 -4600.517,E2 -4600.517} C_VEL
LIN {X 0,Y 524.8,Z 343.225,A -85,B 0,C 180,E1 -4600.83,E2 -4600.83} C_VEL
LIN {X 0,Y 524.873,Z 322.402,A -85,B 0,C 180,E1 -4601.143,E2 -4601.143} C_VEL
LIN {X 0,Y 524.846,Z 273.274,A -85,B 0,C 180,E1 -4601.816,E2 -4601.816} C_VEL
LIN {X 0,Y 523.693,Z 265.933,A -85,B 0,C 180,E1 -4601.962,E2 -4601.962} C_VEL
LIN {X 0,Y 523.71,Z 251.869,A -85,B 0,C 180,E1 -4605.157,E2 -4605.157} C_VEL
LIN {X 0,Y 523.748,Z 250.064,A -85,B 0,C 180,E1 -4605.617,E2 -4605.617} C_VEL
LIN {X 0,Y 523.912,Z 250.036,A -85,B 0,C 180,E1 -4607.97,E2 -4607.97} C_VEL
LIN {X 0,Y 523.941,Z 250.03,A -85,B 0,C 180,E1 -4610.411,E2 -4610.411} C_VEL
LIN {X 0,Y 523.883,Z 250.04,A -85,B 0,C 180,E1 -4612.894,E2 -4612.894} C_VEL
LIN {X 0,Y 523.896,Z 250.041,A -85,B 0,C 180,E1 -4615.421,E2 -4615.421} C_VEL
LIN {X 0,Y 523.895,Z 250.036,A -85,B 0,C 180,E1 -4618.003,E2 -4618.003} C_VEL
LIN {X 0,Y 523.896,Z 250.04,A -85,B 0,C 180,E1 -4620.845,E2 -4620.845} C_VEL
LIN {X 0,Y 523.923,Z 250.034,A -85,B 0,C 180,E1 -4623.728,E2 -4623.728} C_VEL
LIN {X 0,Y 523.884,Z 250.038,A -85,B 0,C 180,E1 -4626.398,E2 -4626.398} C_VEL
LIN {X 0,Y 523.907,Z 250.039,A -85,B 0,C 180,E1 -4629.085,E2 -4629.085} C_VEL
LIN {X 0,Y 523.889,Z 250.037,A -85,B 0,C 180,E1 -4632.124,E2 -4632.124} C_VEL
LIN {X 0,Y 523.93,Z 250.034,A -85,B 0,C 180,E1 -4635.311,E2 -4635.311} C_VEL
LIN {X 0,Y 523.907,Z 250.04,A -85,B 0,C 180,E1 -4638.695,E2 -4638.695} C_VEL
LIN {X 0,Y 523.905,Z 250.035,A -85,B 0,C 180,E1 -4641.897,E2 -4641.897} C_VEL
LIN {X 0,Y 523.91,Z 250.039,A -85,B 0,C 180,E1 -4644.912,E2 -4644.912} C_VEL
LIN {X 0,Y 523.926,Z 250.032,A -85,B 0,C 180,E1 -4647.68,E2 -4647.68} C_VEL
LIN {X 0,Y 523.925,Z 250.038,A -85,B 0,C 180,E1 -4650.681,E2 -4650.681} C_VEL
LIN {X 0,Y 523.893,Z 250.037,A -85,B 0,C 180,E1 -4653.724,E2 -4653.724} C_VEL
LIN {X 0,Y 523.891,Z 250.041,A -85,B 0,C 180,E1 -4656.268,E2 -4656.268} C_VEL
LIN {X 0,Y 523.917,Z 250.037,A -85,B 0,C 180,E1 -4658.765,E2 -4658.765} C_VEL
LIN {X 0,Y 523.919,Z 250.033,A -85,B 0,C 180,E1 -4661.219,E2 -4661.219} C_VEL
LIN {X 0,Y 523.874,Z 250.04,A -85,B 0,C 180,E1 -4663.637,E2 -4663.637} C_VEL
